LIN {X 0,Y 474.756,Z 198.653,A -85,B 0,C 180,E1 -7374.053,E2 -7374.053} C_VEL
LIN {X 0,Y 474.86,Z 198.632,A -85,B 0,C 180,E1 -7377.456,E2 -7377.456} C_VEL
LIN {X 0,Y 474.875,Z 198.64,A -85,B 0,C 180,E1 -7380,E2 -7380} C_VEL
LIN {X 0,Y 474.861,Z 198.647,A -85,B 0,C 180,E1 -7382.545,E2 -7382.545} C_VEL
LIN {X 0,Y 474.75,Z 198.651,A -85,B 0,C 180,E1 -7385.948,E2 -7385.948} C_VEL
LIN {X 0,Y 474.696,Z 198.67,A -85,B 0,C 180,E1 -7388.515,E2 -7388.515} C_VEL
LIN {X 0,Y 474.673,Z 198.655,A -85,B 0,C 180,E1 -7391.964,E2 -7391.964} C_VEL
LIN {X 0,Y 474.669,Z 198.666,A -85,B 0,C 180,E1 -7395.457,E2 -7395.457} C_VEL
LIN {X 0,Y 474.635,Z 198.663,A -85,B 0,C 180,E1 -7399.012,E2 -7399.012} C_VEL
LIN {X 0,Y 474.568,Z 198.678,A -85,B 0,C 180,E1 -7401.73,E2 -7401.73} C_VEL
LIN {X 0,Y 474.634,Z 198.67,A -85,B 0,C 180,E1 -7404.495,E2 -7404.495} C_VEL
LIN {X 0,Y 474.654,Z 198.664,A -85,B 0,C 180,E1 -7407.337,E2 -7407.337} C_VEL
LIN {X 0,Y 474.579,Z 198.684,A -85,B 0,C 180,E1 -7410.233,E2 -7410.233} C_VEL
LIN {X 0,Y 474.618,Z 198.665,A -85,B 0,C 180,E1 -7413.223,E2 -7413.223} C_VEL
LIN {X 0,Y 474.568,Z 198.687,A -85,B 0,C 180,E1 -7416.326,E2 -7416.326} C_VEL
LIN {X 0,Y 474.595,Z 198.667,A -85,B 0,C 180,E1 -7419.649,E2 -7419.649} C_VEL
LIN {X 0,Y 474.604,Z 198.682,A -85,B 0,C 180,E1 -7422.24,E2 -7422.24} C_VEL
LIN {X 0,Y 474.598,Z 198.667,A -85,B 0,C 180,E1 -7425.301,E2 -7425.301} C_VEL
LIN {X 0,Y 474.598,Z 198.682,A -85,B 0,C 180,E1 -7428.217,E2 -7428.217} C_VEL
LIN {X 0,Y 474.597,Z 198.672,A -85,B 0,C 180,E1 -7431.546,E2 -7431.546} C_VEL
LIN {X 0,Y 474.615,Z 198.669,A -85,B 0,C 180,E1 -7434.729,E2 -7434.729} C_VEL
LIN {X 0,Y 474.625,Z 198.676,A -85,B 0,C 180,E1 -7437.791,E2 -7437.791} C_VEL
LIN {X 0,Y 474.598,Z 198.675,A -85,B 0,C 180,E1 -7440.892,E2 -7440.892} C_VEL
LIN {X 0,Y 474.595,Z 198.679,A -85,B 0,C 180,E1 -7443.628,E2 -7443.628} C_VEL
LIN {X 0,Y 474.629,Z 198.672,A -85,B 0,C 180,E1 -7446.645,E2 -7446.645} C_VEL
LIN {X 0,Y 474.644,Z 198.673,A -85,B 0,C 180,E1 -7450.092,E2 -7450.092} C_VEL
LIN {X 0,Y 474.635,Z 198.675,A -85,B 0,C 180,E1 -7451.709,E2 -7451.709} C_VEL
LIN {X 0,Y 473.961,Z 198.765,A -85,B 0,C 180,E1 -7452.418,E2 -7452.418} C_VEL
LIN {X 0,Y 471.109,Z 199.122,A -85,B 0,C 180,E1 -7453.569,E2 -7453.569} C_VEL
LIN {X 0,Y 468.702,Z 199.417,A -85,B 0,C 180,E1 -7454.497,E2 -7454.497} C_VEL
LIN {X 0,Y 467.668,Z 199.542,A -85,B 0,C 180,E1 -7455.214,E2 -7455.214} C_VEL
LIN {X 0,Y 467.584,Z 199.551,A -85,B 0,C 180,E1 -7455.457,E2 -7455.457} C_VEL
LIN {X 0,Y 467.65,Z 199.543,A -85,B 0,C 180,E1 -7458.736,E2 -7458.736} C_VEL
LIN {X 0,Y 467.658,Z 199.545,A -85,B 0,C 180,E1 -7461.359,E2 -7461.359} C_VEL
LIN {X 0,Y 467.705,Z 199.531,A -85,B 0,C 180,E1 -7463.964,E2 -7463.964} C_VEL
LIN {X 0,Y 467.597,Z 199.662,A -85,B 0,C 180,E1 -7466.367,E2 -7466.367} C_VEL
LIN {X 0,Y 470.549,Z 209.002,A -85,B 0,C 180,E1 -7467.722,E2 -7467.722} C_VEL
LIN {X 0,Y 480.125,Z 229.823,A -85,B 0,C 180,E1 -7468.71,E2 -7468.71} C_VEL
LIN {X 0,Y 478.57,Z 337.497,A -85,B 0,C 180,E1 -7470.42,E2 -7470.42} C_VEL
LIN {X 0,Y 477.488,Z 414.636,A -85,B 0,C 180,E1 -7471.66,E2 -7471.66} C_VEL
LIN {X 0,Y 476.912,Z 431.039,A -85,B 0,C 180,E1 -7472.087,E2 -7472.087} C_VEL
LIN {X 0,Y 476.258,Z 446.341,A -85,B 0,C 180,E1 -7472.645,E2 -7472.645} C_VEL
LIN {X 0,Y 475.341,Z 462.22,A -85,B 0,C 180,E1 -7473.392,E2 -7473.392} C_VEL
LIN {X 0,Y 474.435,Z 476.76,A -85,B 0,C 180,E1 -7474.249,E2 -7474.249} C_VEL
LIN {X 0,Y 473.289,Z 491.411,A -85,B 0,C 180,E1 -7475.302,E2 -7475.302} C_VEL
LIN {X 0,Y 472.273,Z 504.308,A -85,B 0,C 180,E1 -7476.41,E2 -7476.41} C_VEL
LIN {X 0,Y 471.217,Z 517.245,A -85,B 0,C 180,E1 -7477.716,E2 -7477.716} C_VEL
LIN {X 0,Y 470.216,Z 529.305,A -85,B 0,C 180,E1 -7479.147,E2 -7479.147} C_VEL
LIN {X 0,Y 469.224,Z 540.984,A -85,B 0,C 180,E1 -7480.792,E2 -7480.792} C_VEL
LIN {X 0,Y 468.482,Z 550.373,A -85,B 0,C 180,E1 -7482.355,E2 -7482.355} C_VEL
LIN {X 0,Y 467.914,Z 559.42,A -85,B 0,C 180,E1 -7484.129,E2 -7484.129} C_VEL
LIN {X 0,Y 467.444,Z 566.588,A -85,B 0,C 180,E1 -7485.794,E2 -7485.794} C_VEL
LIN {X 0,Y 467.03,Z 574.14,A -85,B 0,C 180,E1 -7487.97,E2 -7487.97} C_VEL
LIN {X 0,Y 466.828,Z 579.053,A -85,B 0,C 180,E1 -7489.801,E2 -7489.801} C_VEL
LIN {X 0,Y 466.675,Z 582.05,A -85,B 0,C 180,E1 -7491.19,E2 -7491.19} C_VEL
LIN {X 0,Y 466.513,Z 585.196,A -85,B 0,C 180,E1 -7493.224,E2 -7493.224} C_VEL
LIN {X 0,Y 466.473,Z 587.043,A -85,B 0,C 180,E1 -7495.313,E2 -7495.313} C_VEL
LIN {X 0,Y 466.497,Z 587.539,A -85,B 0,C 180,E1 -7497.268,E2 -7497.268} C_VEL
LIN {X 0,Y 466.524,Z 586.882,A -85,B 0,C 180,E1 -7499.102,E2 -7499.102} C_VEL
LIN {X 0,Y 466.589,Z 585.259,A -85,B 0,C 180,E1 -7500.843,E2 -7500.843} C_VEL
LIN {X 0,Y 466.678,Z 582.245,A -85,B 0,C 180,E1 -7502.831,E2 -7502.831} C_VEL
LIN {X 0,Y 466.811,Z 579.574,A -85,B 0,C 180,E1 -7504.101,E2 -7504.101} C_VEL
LIN {X 0,Y 467.041,Z 574.75,A -85,B 0,C 180,E1 -7505.936,E2 -7505.936} C_VEL
LIN {X 0,Y 467.282,Z 569.408,A -85,B 0,C 180,E1 -7507.562,E2 -7507.562} C_VEL
LIN {X 0,Y 467.669,Z 563.253,A -85,B 0,C 180,E1 -7509.137,E2 -7509.137} C_VEL
LIN {X 0,Y 468.147,Z 555.633,A -85,B 0,C 180,E1 -7510.772,E2 -7510.772} C_VEL
LIN {X 0,Y 468.822,Z 546.607,A -85,B 0,C 180,E1 -7512.423,E2 -7512.423} C_VEL
LIN {X 0,Y 469.752,Z 535.757,A -85,B 0,C 180,E1 -7514.099,E2 -7514.099} C_VEL
LIN {X 0,Y 470.651,Z 524.675,A -85,B 0,C 180,E1 -7515.547,E2 -7515.547} C_VEL
LIN {X 0,Y 471.687,Z 512.615,A -85,B 0,C 180,E1 -7516.894,E2 -7516.894} C_VEL
LIN {X 0,Y 472.776,Z 499.201,A -85,B 0,C 180,E1 -7518.171,E2 -7518.171} C_VEL
LIN {X 0,Y 473.863,Z 485.577,A -85,B 0,C 180,E1 -7519.263,E2 -7519.263} C_VEL
LIN {X 0,Y 474.967,Z 469.802,A -85,B 0,C 180,E1 -7520.304,E2 -7520.304} C_VEL
LIN {X 0,Y 475.881,Z 455.142,A -85,B 0,C 180,E1 -7521.081,E2 -7521.081} C_VEL
LIN {X 0,Y 476.692,Z 438.798,A -85,B 0,C 180,E1 -7521.767,E2 -7521.767} C_VEL
LIN {X 0,Y 477.372,Z 422.454,A -85,B 0,C 180,E1 -7522.269,E2 -7522.269} C_VEL
LIN {X 0,Y 477.774,Z 405.589,A -85,B 0,C 180,E1 -7522.617,E2 -7522.617} C_VEL
LIN {X 0,Y 480.45,Z 230.253,A -85,B 0,C 180,E1 -7525.405,E2 -7525.405} C_VEL
LIN {X 0,Y 471.765,Z 211.838,A -85,B 0,C 180,E1 -7526.32,E2 -7526.32} C_VEL
LIN {X 0,Y 470.58,Z 209.292,A -85,B 0,C 180,E1 -7526.455,E2 -7526.455} C_VEL
LIN {X 0,Y 467.6,Z 199.551,A -85,B 0,C 180,E1 -7527.944,E2 -7527.944} C_VEL
LIN {X 0,Y 467.579,Z 199.553,A -85,B 0,C 180,E1 -7531.25,E2 -7531.25} C_VEL
LIN {X 0,Y 467.599,Z 199.551,A -85,B 0,C 180,E1 -7534.159,E2 -7534.159} C_VEL
LIN {X 0,Y 467.577,Z 199.554,A -85,B 0,C 180,E1 -7536.995,E2 -7536.995} C_VEL
LIN {X 0,Y 467.624,Z 199.545,A -85,B 0,C 180,E1 -7539.777,E2 -7539.777} C_VEL
LIN {X 0,Y 467.609,Z 199.543,A -85,B 0,C 180,E1 -7542.506,E2 -7542.506} C_VEL
LIN {X 0,Y 467.606,Z 199.548,A -85,B 0,C 180,E1 -7545.196,E2 -7545.196} C_VEL
LIN {X 0,Y 467.656,Z 199.546,A -85,B 0,C 180,E1 -7547.854,E2 -7547.854} C_VEL
LIN {X 0,Y 467.679,Z 199.541,A -85,B 0,C 180,E1 -7551.357,E2 -7551.357} C_VEL
LIN {X 0,Y 467.741,Z 199.534,A -85,B 0,C 180,E1 -7553.962,E2 -7553.962} C_VEL
LIN {X 0,Y 467.856,Z 199.518,A -85,B 0,C 180,E1 -7557.417,E2 -7557.417} C_VEL
LIN {X 0,Y 467.879,Z 199.518,A -85,B 0,C 180,E1 -7560,E2 -7560} C_VEL
LIN {X 0,Y 467.855,Z 199.516,A -85,B 0,C 180,E1 -7562.582,E2 -7562.582} C_VEL
LIN {X 0,Y 467.731,Z 199.534,A -85,B 0,C 180,E1 -7566.037,E2 -7566.037} C_VEL
LIN {X 0,Y 467.668,Z 199.54,A -85,B 0,C 180,E1 -7568.643,E2 -7568.643} C_VEL
LIN {X 0,Y 467.654,Z 199.542,A -85,B 0,C 180,E1 -7572.145,E2 -7572.145} C_VEL
LIN {X 0,Y 467.637,Z 199.545,A -85,B 0,C 180,E1 -7575.695,E2 -7575.695} C_VEL
LIN {X 0,Y 467.62,Z 199.548,A -85,B 0,C 180,E1 -7579.307,E2 -7579.307} C_VEL
LIN {X 0,Y 467.532,Z 199.556,A -85,B 0,C 180,E1 -7582.074,E2 -7582.074} C_VEL
LIN {X 0,Y 467.583,Z 199.55,A -85,B 0,C 180,E1 -7584.888,E2 -7584.888} C_VEL
LIN {X 0,Y 467.618,Z 199.548,A -85,B 0,C 180,E1 -7587.769,E2 -7587.769} C_VEL
LIN {X 0,Y 467.566,Z 199.558,A -85,B 0,C 180,E1 -7591.044,E2 -7591.044} C_VEL
LIN {X 0,Y 467.576,Z 199.55,A -85,B 0,C 180,E1 -7594.239,E2 -7594.239} C_VEL
LIN {X 0,Y 467.547,Z 199.561,A -85,B 0,C 180,E1 -7597.186,E2 -7597.186} C_VEL
LIN {X 0,Y 467.57,Z 199.552,A -85,B 0,C 180,E1 -7600.265,E2 -7600.265} C_VEL
LIN {X 0,Y 467.548,Z 199.555,A -85,B 0,C 180,E1 -7603.745,E2 -7603.745} C_VEL
LIN {X 0,Y 467.547,Z 199.56,A -85,B 0,C 180,E1 -7606.254,E2 -7606.254} C_VEL
LIN {X 0,Y 467.56,Z 199.555,A -85,B 0,C 180,E1 -7609.733,E2 -7609.733} C_VEL
LIN {X 0,Y 467.543,Z 199.557,A -85,B 0,C 180,E1 -7612.814,E2 -7612.814} C_VEL
LIN {X 0,Y 467.585,Z 199.552,A -85,B 0,C 180,E1 -7616.211,E2 -7616.211} C_VEL
LIN {X 0,Y 467.622,Z 199.679,A -85,B 0,C 180,E1 -7616.715,E2 -7616.715} C_VEL
LIN {X 0,Y 473.66,Z 219.016,A -85,B 0,C 180,E1 -7619.381,E2 -7619.381} C_VEL
LIN {X 0,Y 475.873,Z 227.663,A -85,B 0,C 180,E1 -7620.491,E2 -7620.491} C_VEL
LIN {X 0,Y 475.592,Z 231.809,A -85,B 0,C 180,E1 -7620.928,E2 -7620.928} C_VEL
LIN {X 0,Y 480.062,Z 257.211,A -85,B 0,C 180,E1 -7621.668,E2 -7621.668} C_VEL
LIN {X 0,Y 478.274,Z 376.342,A -85,B 0,C 180,E1 -7623.564,E2 -7623.564} C_VEL
LIN {X 0,Y 477.338,Z 440.054,A -85,B 0,C 180,E1 -7624.595,E2 -7624.595} C_VEL
LIN {X 0,Y 476.616,Z 457.299,A -85,B 0,C 180,E1 -7625.047,E2 -7625.047} C_VEL
LIN {X 0,Y 475.877,Z 472.946,A -85,B 0,C 180,E1 -7625.631,E2 -7625.631} C_VEL
LIN {X 0,Y 474.949,Z 487.77,A -85,B 0,C 180,E1 -7626.334,E2 -7626.334} C_VEL
LIN {X 0,Y 473.975,Z 502.298,A -85,B 0,C 180,E1 -7627.187,E2 -7627.187} C_VEL
LIN {X 0,Y 472.892,Z 516.304,A -85,B 0,C 180,E1 -7628.188,E2 -7628.188} C_VEL
LIN {X 0,Y 471.72,Z 530.44,A -85,B 0,C 180,E1 -7629.39,E2 -7629.39} C_VEL
LIN {X 0,Y 470.682,Z 542.772,A -85,B 0,C 180,E1 -7630.625,E2 -7630.625} C_VEL
LIN {X 0,Y 469.688,Z 555.582,A -85,B 0,C 180,E1 -7632.135,E2 -7632.135} C_VEL
LIN {X 0,Y 468.773,Z 567.224,A -85,B 0,C 180,E1 -7633.762,E2 -7633.762} C_VEL
LIN {X 0,Y 468.157,Z 576.066,A -85,B 0,C 180,E1 -7635.213,E2 -7635.213} C_VEL
LIN {X 0,Y 467.611,Z 585.271,A -85,B 0,C 180,E1 -7636.969,E2 -7636.969} C_VEL
LIN {X 0,Y 467.2,Z 592.974,A -85,B 0,C 180,E1 -7638.721,E2 -7638.721} C_VEL
LIN {X 0,Y 466.853,Z 600.714,A -85,B 0,C 180,E1 -7640.904,E2 -7640.904} C_VEL
LIN {X 0,Y 466.772,Z 605.522,A -85,B 0,C 180,E1 -7642.645,E2 -7642.645} C_VEL
LIN {X 0,Y 466.697,Z 608.448,A -85,B 0,C 180,E1 -7643.947,E2 -7643.947} C_VEL
LIN {X 0,Y 466.599,Z 611.421,A -85,B 0,C 180,E1 -7645.679,E2 -7645.679} C_VEL
LIN {X 0,Y 466.651,Z 613.381,A -85,B 0,C 180,E1 -7647.408,E2 -7647.408} C_VEL
LIN {X 0,Y 466.615,Z 614.357,A -85,B 0,C 180,E1 -7649.135,E2 -7649.135} C_VEL
LIN {X 0,Y 466.615,Z 614.365,A -85,B 0,C 180,E1 -7650.861,E2 -7650.861} C_VEL
LIN {X 0,Y 466.65,Z 613.404,A -85,B 0,C 180,E1 -7652.587,E2 -7652.587} C_VEL
LIN {X 0,Y 466.598,Z 611.461,A -85,B 0,C 180,E1 -7654.317,E2 -7654.317} C_VEL
LIN {X 0,Y 466.746,Z 607.794,A -85,B 0,C 180,E1 -7656.391,E2 -7656.391} C_VEL
LIN {X 0,Y 466.79,Z 603.336,A -85,B 0,C 180,E1 -7658.221,E2 -7658.221} C_VEL
LIN {X 0,Y 466.969,Z 597.932,A -85,B 0,C 180,E1 -7659.964,E2 -7659.964} C_VEL
LIN {X 0,Y 467.336,Z 591.264,A -85,B 0,C 180,E1 -7661.711,E2 -7661.711} C_VEL
LIN {X 0,Y 467.733,Z 583.271,A -85,B 0,C 180,E1 -7663.465,E2 -7663.465} C_VEL
LIN {X 0,Y 468.419,Z 573.731,A -85,B 0,C 180,E1 -7665.22,E2 -7665.22} C_VEL
LIN {X 0,Y 469.184,Z 562.298,A -85,B 0,C 180,E1 -7666.981,E2 -7666.981} C_VEL
LIN {X 0,Y 470.161,Z 550.414,A -85,B 0,C 180,E1 -7668.518,E2 -7668.518} C_VEL
LIN {X 0,Y 471.123,Z 538.265,A -85,B 0,C 180,E1 -7669.861,E2 -7669.861} C_VEL
LIN {X 0,Y 472.265,Z 524.529,A -85,B 0,C 180,E1 -7671.151,E2 -7671.151} C_VEL
LIN {X 0,Y 473.318,Z 510.73,A -85,B 0,C 180,E1 -7672.246,E2 -7672.246} C_VEL
LIN {X 0,Y 474.473,Z 494.982,A -85,B 0,C 180,E1 -7673.27,E2 -7673.27} C_VEL
LIN {X 0,Y 475.417,Z 480.293,A -85,B 0,C 180,E1 -7674.042,E2 -7674.042} C_VEL
LIN {X 0,Y 476.317,Z 463.971,A -85,B 0,C 180,E1 -7674.718,E2 -7674.718} C_VEL
LIN {X 0,Y 476.985,Z 448.256,A -85,B 0,C 180,E1 -7675.205,E2 -7675.205} C_VEL
LIN {X 0,Y 477.512,Z 431.69,A -85,B 0,C 180,E1 -7675.546,E2 -7675.546} C_VEL
LIN {X 0,Y 479.984,Z 258.583,A -85,B 0,C 180,E1 -7678.281,E2 -7678.281} C_VEL
LIN {X 0,Y 478.559,Z 248.971,A -85,B 0,C 180,E1 -7678.534,E2 -7678.534} C_VEL
LIN {X 0,Y 475.596,Z 232.132,A -85,B 0,C 180,E1 -7679.039,E2 -7679.039} C_VEL
LIN {X 0,Y 475.884,Z 227.612,A -85,B 0,C 180,E1 -7679.514,E2 -7679.514} C_VEL
LIN {X 0,Y 472.324,Z 214.704,A -85,B 0,C 180,E1 -7681.178,E2 -7681.178} C_VEL
LIN {X 0,Y 467.604,Z 199.536,A -85,B 0,C 180,E1 -7683.266,E2 -7683.266} C_VEL
LIN {X 0,Y 467.536,Z 199.56,A -85,B 0,C 180,E1 -7685.887,E2 -7685.887} C_VEL
LIN {X 0,Y 467.556,Z 199.559,A -85,B 0,C 180,E1 -7689.143,E2 -7689.143} C_VEL
LIN {X 0,Y 467.565,Z 199.552,A -85,B 0,C 180,E1 -7692.565,E2 -7692.565} C_VEL
LIN {X 0,Y 467.547,Z 199.556,A -85,B 0,C 180,E1 -7695.051,E2 -7695.051} C_VEL
LIN {X 0,Y 467.565,Z 199.557,A -85,B 0,C 180,E1 -7697.438,E2 -7697.438} C_VEL
LIN {X 0,Y 467.587,Z 199.553,A -85,B 0,C 180,E1 -7700.856,E2 -7700.856} C_VEL
LIN {X 0,Y 467.535,Z 199.552,A -85,B 0,C 180,E1 -7704.258,E2 -7704.258} C_VEL
LIN {X 0,Y 467.554,Z 199.548,A -85,B 0,C 180,E1 -7707.319,E2 -7707.319} C_VEL
LIN {X 0,Y 467.54,Z 199.559,A -85,B 0,C 180,E1 -7710.666,E2 -7710.666} C_VEL
LIN {X 0,Y 467.585,Z 199.542,A -85,B 0,C 180,E1 -7713.198,E2 -7713.198} C_VEL
LIN {X 0,Y 467.566,Z 199.554,A -85,B 0,C 180,E1 -7716.466,E2 -7716.466} C_VEL
LIN {X 0,Y 467.594,Z 199.536,A -85,B 0,C 180,E1 -7719.776,E2 -7719.776} C_VEL
LIN {X 0,Y 467.576,Z 199.549,A -85,B 0,C 180,E1 -7722.506,E2 -7722.506} C_VEL
LIN {X 0,Y 467.573,Z 199.549,A -85,B 0,C 180,E1 -7725.196,E2 -7725.196} C_VEL
LIN {X 0,Y 467.65,Z 199.521,A -85,B 0,C 180,E1 -7727.855,E2 -7727.855} C_VEL
LIN {X 0,Y 467.65,Z 199.543,A -85,B 0,C 180,E1 -7731.357,E2 -7731.357} C_VEL
LIN {X 0,Y 467.718,Z 199.529,A -85,B 0,C 180,E1 -7733.963,E2 -7733.963} C_VEL
LIN {X 0,Y 467.826,Z 199.508,A -85,B 0,C 180,E1 -7737.417,E2 -7737.417} C_VEL
LIN {X 0,Y 467.846,Z 199.516,A -85,B 0,C 180,E1 -7740,E2 -7740} C_VEL
LIN {X 0,Y 467.826,Z 199.522,A -85,B 0,C 180,E1 -7742.584,E2 -7742.584} C_VEL
LIN {X 0,Y 467.714,Z 199.528,A -85,B 0,C 180,E1 -7746.038,E2 -7746.038} C_VEL
LIN {X 0,Y 467.65,Z 199.546,A -85,B 0,C 180,E1 -7748.644,E2 -7748.644} C_VEL
LIN {X 0,Y 467.624,Z 199.534,A -85,B 0,C 180,E1 -7752.147,E2 -7752.147} C_VEL
LIN {X 0,Y 467.624,Z 199.544,A -85,B 0,C 180,E1 -7755.696,E2 -7755.696} C_VEL
LIN {X 0,Y 467.587,Z 199.541,A -85,B 0,C 180,E1 -7758.766,E2 -7758.766} C_VEL
LIN {X 0,Y 467.554,Z 199.552,A -85,B 0,C 180,E1 -7761.271,E2 -7761.271} C_VEL
LIN {X 0,Y 467.547,Z 199.555,A -85,B 0,C 180,E1 -7763.945,E2 -7763.945} C_VEL
LIN {X 0,Y 467.589,Z 199.547,A -85,B 0,C 180,E1 -7766.803,E2 -7766.803} C_VEL
LIN {X 0,Y 467.527,Z 199.558,A -85,B 0,C 180,E1 -7769.741,E2 -7769.741} C_VEL
LIN {X 0,Y 467.558,Z 199.546,A -85,B 0,C 180,E1 -7772.761,E2 -7772.761} C_VEL
LIN {X 0,Y 467.532,Z 199.558,A -85,B 0,C 180,E1 -7775.892,E2 -7775.892} C_VEL
LIN {X 0,Y 467.537,Z 199.544,A -85,B 0,C 180,E1 -7779.15,E2 -7779.15} C_VEL
LIN {X 0,Y 467.567,Z 199.555,A -85,B 0,C 180,E1 -7782.57,E2 -7782.57} C_VEL
LIN {X 0,Y 467.547,Z 199.545,A -85,B 0,C 180,E1 -7785.055,E2 -7785.055} C_VEL
LIN {X 0,Y 467.557,Z 199.554,A -85,B 0,C 180,E1 -7788.6,E2 -7788.6} C_VEL
LIN {X 0,Y 467.551,Z 199.554,A -85,B 0,C 180,E1 -7791.959,E2 -7791.959} C_VEL
LIN {X 0,Y 467.554,Z 199.547,A -85,B 0,C 180,E1 -7795.171,E2 -7795.171} C_VEL
LIN {X 0,Y 467.572,Z 199.556,A -85,B 0,C 180,E1 -7798.263,E2 -7798.263} C_VEL
LIN {X 0,Y 467.546,Z 199.553,A -85,B 0,C 180,E1 -7801.252,E2 -7801.252} C_VEL
LIN {X 0,Y 467.572,Z 199.552,A -85,B 0,C 180,E1 -7804.161,E2 -7804.161} C_VEL
LIN {X 0,Y 467.57,Z 199.55,A -85,B 0,C 180,E1 -7806.999,E2 -7806.999} C_VEL
LIN {X 0,Y 467.615,Z 199.553,A -85,B 0,C 180,E1 -7809.78,E2 -7809.78} C_VEL
LIN {X 0,Y 467.565,Z 199.555,A -85,B 0,C 180,E1 -7812.508,E2 -7812.508} C_VEL
LIN {X 0,Y 467.584,Z 199.551,A -85,B 0,C 180,E1 -7815.457,E2 -7815.457} C_VEL
LIN {X 0,Y 466.918,Z 199.636,A -85,B 0,C 180,E1 -7816.176,E2 -7816.176} C_VEL
LIN {X 0,Y 464.078,Z 199.99,A -85,B 0,C 180,E1 -7817.345,E2 -7817.345} C_VEL
LIN {X 0,Y 461.68,Z 200.288,A -85,B 0,C 180,E1 -7818.287,E2 -7818.287} C_VEL
LIN {X 0,Y 460.653,Z 200.415,A -85,B 0,C 180,E1 -7819.015,E2 -7819.015} C_VEL
LIN {X 0,Y 460.571,Z 200.426,A -85,B 0,C 180,E1 -7819.261,E2 -7819.261} C_VEL
LIN {X 0,Y 460.666,Z 200.416,A -85,B 0,C 180,E1 -7822.596,E2 -7822.596} C_VEL
LIN {X 0,Y 460.677,Z 200.403,A -85,B 0,C 180,E1 -7824.75,E2 -7824.75} C_VEL
LIN {X 0,Y 460.553,Z 200.62,A -85,B 0,C 180,E1 -7825.955,E2 -7825.955} C_VEL
LIN {X 0,Y 463.312,Z 209.012,A -85,B 0,C 180,E1 -7827.225,E2 -7827.225} C_VEL
LIN {X 0,Y 473.85,Z 231.782,A -85,B 0,C 180,E1 -7828.337,E2 -7828.337} C_VEL
LIN {X 0,Y 472.34,Z 332.526,A -85,B 0,C 180,E1 -7829.962,E2 -7829.962} C_VEL
LIN {X 0,Y 471.041,Z 415.463,A -85,B 0,C 180,E1 -7831.311,E2 -7831.311} C_VEL
LIN {X 0,Y 470.43,Z 432.452,A -85,B 0,C 180,E1 -7831.768,E2 -7831.768} C_VEL
LIN {X 0,Y 469.701,Z 448.061,A -85,B 0,C 180,E1 -7832.36,E2 -7832.36} C_VEL
LIN {X 0,Y 468.723,Z 463.616,A -85,B 0,C 180,E1 -7833.118,E2 -7833.118} C_VEL
LIN {X 0,Y 467.764,Z 477.967,A -85,B 0,C 180,E1 -7833.987,E2 -7833.987} C_VEL
LIN {X 0,Y 466.566,Z 492.8,A -85,B 0,C 180,E1 -7835.079,E2 -7835.079} C_VEL
LIN {X 0,Y 465.442,Z 506.377,A -85,B 0,C 180,E1 -7836.287,E2 -7836.287} C_VEL
LIN {X 0,Y 464.298,Z 519.039,A -85,B 0,C 180,E1 -7837.613,E2 -7837.613} C_VEL
LIN {X 0,Y 463.321,Z 530.181,A -85,B 0,C 180,E1 -7838.973,E2 -7838.973} C_VEL
LIN {X 0,Y 462.372,Z 540.923,A -85,B 0,C 180,E1 -7840.511,E2 -7840.511} C_VEL
LIN {X 0,Y 461.575,Z 550.304,A -85,B 0,C 180,E1 -7842.086,E2 -7842.086} C_VEL
LIN {X 0,Y 460.928,Z 559.45,A -85,B 0,C 180,E1 -7843.897,E2 -7843.897} C_VEL
LIN {X 0,Y 460.452,Z 566.134,A -85,B 0,C 180,E1 -7845.463,E2 -7845.463} C_VEL
LIN {X 0,Y 460.041,Z 572.746,A -85,B 0,C 180,E1 -7847.333,E2 -7847.333} C_VEL
LIN {X 0,Y 459.826,Z 578.038,A -85,B 0,C 180,E1 -7849.186,E2 -7849.186} C_VEL
LIN {X 0,Y 459.592,Z 582.296,A -85,B 0,C 180,E1 -7851.123,E2 -7851.123} C_VEL
LIN {X 0,Y 459.435,Z 584.534,A -85,B 0,C 180,E1 -7852.485,E2 -7852.485} C_VEL
LIN {X 0,Y 459.375,Z 586.654,A -85,B 0,C 180,E1 -7854.399,E2 -7854.399} C_VEL
LIN {X 0,Y 459.372,Z 587.654,A -85,B 0,C 180,E1 -7856.34,E2 -7856.34} C_VEL
LIN {X 0,Y 459.413,Z 587.529,A -85,B 0,C 180,E1 -7858.31,E2 -7858.31} C_VEL
LIN {X 0,Y 459.456,Z 586.119,A -85,B 0,C 180,E1 -7860.318,E2 -7860.318} C_VEL
LIN {X 0,Y 459.542,Z 583.383,A -85,B 0,C 180,E1 -7862.363,E2 -7862.363} C_VEL
LIN {X 0,Y 459.748,Z 579.221,A -85,B 0,C 180,E1 -7864.445,E2 -7864.445} C_VEL
LIN {X 0,Y 460.052,Z 573.451,A -85,B 0,C 180,E1 -7866.57,E2 -7866.57} C_VEL
LIN {X 0,Y 460.422,Z 566.932,A -85,B 0,C 180,E1 -7868.465,E2 -7868.465} C_VEL
LIN {X 0,Y 460.963,Z 559.007,A -85,B 0,C 180,E1 -7870.33,E2 -7870.33} C_VEL
LIN {X 0,Y 461.624,Z 550.21,A -85,B 0,C 180,E1 -7872.058,E2 -7872.058} C_VEL
LIN {X 0,Y 462.534,Z 540.105,A -85,B 0,C 180,E1 -7873.738,E2 -7873.738} C_VEL
LIN {X 0,Y 463.467,Z 528.983,A -85,B 0,C 180,E1 -7875.314,E2 -7875.314} C_VEL
LIN {X 0,Y 464.666,Z 516.026,A -85,B 0,C 180,E1 -7876.86,E2 -7876.86} C_VEL
LIN {X 0,Y 465.903,Z 502.305,A -85,B 0,C 180,E1 -7878.23,E2 -7878.23} C_VEL
LIN {X 0,Y 467.106,Z 487.756,A -85,B 0,C 180,E1 -7879.443,E2 -7879.443} C_VEL
LIN {X 0,Y 468.235,Z 473.076,A -85,B 0,C 180,E1 -7880.455,E2 -7880.455} C_VEL
LIN {X 0,Y 469.238,Z 457.631,A -85,B 0,C 180,E1 -7881.325,E2 -7881.325} C_VEL
LIN {X 0,Y 470.082,Z 443.266,A -85,B 0,C 180,E1 -7881.972,E2 -7881.972} C_VEL
LIN {X 0,Y 470.812,Z 426.598,A -85,B 0,C 180,E1 -7882.535,E2 -7882.535} C_VEL
LIN {X 0,Y 471.289,Z 410.62,A -85,B 0,C 180,E1 -7882.905,E2 -7882.905} C_VEL
LIN {X 0,Y 474.22,Z 232.357,A -85,B 0,C 180,E1 -7885.789,E2 -7885.789} C_VEL
LIN {X 0,Y 465.202,Z 213.206,A -85,B 0,C 180,E1 -7886.767,E2 -7886.767} C_VEL
LIN {X 0,Y 463.377,Z 209.586,A -85,B 0,C 180,E1 -7886.971,E2 -7886.971} C_VEL
LIN {X 0,Y 460.549,Z 200.43,A -85,B 0,C 180,E1 -7888.409,E2 -7888.409} C_VEL
LIN {X 0,Y 460.555,Z 200.427,A -85,B 0,C 180,E1 -7891.767,E2 -7891.767} C_VEL
LIN {X 0,Y 460.541,Z 200.434,A -85,B 0,C 180,E1 -7894.704,E2 -7894.704} C_VEL
LIN {X 0,Y 460.512,Z 200.436,A -85,B 0,C 180,E1 -7897.571,E2 -7897.571} C_VEL
LIN {X 0,Y 460.57,Z 200.43,A -85,B 0,C 180,E1 -7900.384,E2 -7900.384} C_VEL
LIN {X 0,Y 460.566,Z 200.421,A -85,B 0,C 180,E1 -7903.146,E2 -7903.146} C_VEL
LIN {X 0,Y 460.554,Z 200.43,A -85,B 0,C 180,E1 -7905.867,E2 -7905.867} C_VEL
LIN {X 0,Y 460.609,Z 200.42,A -85,B 0,C 180,E1 -7908.559,E2 -7908.559} C_VEL
LIN {X 0,Y 460.695,Z 200.414,A -85,B 0,C 180,E1 -7912.108,E2 -7912.108} C_VEL
LIN {X 0,Y 460.694,Z 200.409,A -85,B 0,C 180,E1 -7914.748,E2 -7914.748} C_VEL
LIN {X 0,Y 460.797,Z 200.397,A -85,B 0,C 180,E1 -7917.377,E2 -7917.377} C_VEL
LIN {X 0,Y 460.85,Z 200.394,A -85,B 0,C 180,E1 -7920,E2 -7920} C_VEL
LIN {X 0,Y 460.797,Z 200.396,A -85,B 0,C 180,E1 -7922.622,E2 -7922.622} C_VEL
LIN {X 0,Y 460.696,Z 200.41,A -85,B 0,C 180,E1 -7926.13,E2 -7926.13} C_VEL
LIN {X 0,Y 460.618,Z 200.418,A -85,B 0,C 180,E1 -7928.776,E2 -7928.776} C_VEL
LIN {X 0,Y 460.607,Z 200.419,A -85,B 0,C 180,E1 -7932.334,E2 -7932.334} C_VEL
LIN {X 0,Y 460.6,Z 200.42,A -85,B 0,C 180,E1 -7935.997,E2 -7935.997} C_VEL
LIN {X 0,Y 460.566,Z 200.429,A -85,B 0,C 180,E1 -7939.615,E2 -7939.615} C_VEL
LIN {X 0,Y 460.508,Z 200.43,A -85,B 0,C 180,E1 -7942.428,E2 -7942.428} C_VEL
LIN {X 0,Y 460.551,Z 200.428,A -85,B 0,C 180,E1 -7945.797,E2 -7945.797} C_VEL
LIN {X 0,Y 460.55,Z 200.427,A -85,B 0,C 180,E1 -7948.233,E2 -7948.233} C_VEL
LIN {X 0,Y 460.519,Z 200.434,A -85,B 0,C 180,E1 -7951.282,E2 -7951.282} C_VEL
LIN {X 0,Y 460.522,Z 200.429,A -85,B 0,C 180,E1 -7954.503,E2 -7954.503} C_VEL
LIN {X 0,Y 460.5,Z 200.434,A -85,B 0,C 180,E1 -7957.623,E2 -7957.623} C_VEL
LIN {X 0,Y 460.534,Z 200.429,A -85,B 0,C 180,E1 -7960.268,E2 -7960.268} C_VEL
LIN {X 0,Y 460.508,Z 200.435,A -85,B 0,C 180,E1 -7963.374,E2 -7963.374} C_VEL
LIN {X 0,Y 460.503,Z 200.44,A -85,B 0,C 180,E1 -7966.624,E2 -7966.624} C_VEL
LIN {X 0,Y 460.526,Z 200.431,A -85,B 0,C 180,E1 -7969.732,E2 -7969.732} C_VEL
LIN {X 0,Y 460.497,Z 200.434,A -85,B 0,C 180,E1 -7972.524,E2 -7972.524} C_VEL
LIN {X 0,Y 460.547,Z 200.431,A -85,B 0,C 180,E1 -7975.623,E2 -7975.623} C_VEL
LIN {X 0,Y 460.578,Z 200.535,A -85,B 0,C 180,E1 -7976.246,E2 -7976.246} C_VEL
LIN {X 0,Y 466.068,Z 217.829,A -85,B 0,C 180,E1 -7978.705,E2 -7978.705} C_VEL
LIN {X 0,Y 469.121,Z 228.633,A -85,B 0,C 180,E1 -7980.148,E2 -7980.148} C_VEL
LIN {X 0,Y 469.178,Z 231.798,A -85,B 0,C 180,E1 -7980.49,E2 -7980.49} C_VEL
LIN {X 0,Y 473.834,Z 258.34,A -85,B 0,C 180,E1 -7981.276,E2 -7981.276} C_VEL
LIN {X 0,Y 472.131,Z 363.89,A -85,B 0,C 180,E1 -7982.979,E2 -7982.979} C_VEL
LIN {X 0,Y 470.97,Z 438.936,A -85,B 0,C 180,E1 -7984.206,E2 -7984.206} C_VEL
LIN {X 0,Y 470.23,Z 455.754,A -85,B 0,C 180,E1 -7984.64,E2 -7984.64} C_VEL
LIN {X 0,Y 469.455,Z 471.44,A -85,B 0,C 180,E1 -7985.216,E2 -7985.216} C_VEL
LIN {X 0,Y 468.387,Z 487.561,A -85,B 0,C 180,E1 -7985.982,E2 -7985.982} C_VEL
LIN {X 0,Y 467.385,Z 502.31,A -85,B 0,C 180,E1 -7986.862,E2 -7986.862} C_VEL
LIN {X 0,Y 466.191,Z 516.083,A -85,B 0,C 180,E1 -7987.858,E2 -7987.858} C_VEL
LIN {X 0,Y 464.965,Z 530.214,A -85,B 0,C 180,E1 -7989.077,E2 -7989.077} C_VEL
LIN {X 0,Y 463.889,Z 542.737,A -85,B 0,C 180,E1 -7990.351,E2 -7990.351} C_VEL
LIN {X 0,Y 462.821,Z 555.359,A -85,B 0,C 180,E1 -7991.861,E2 -7991.861} C_VEL
LIN {X 0,Y 461.878,Z 566.634,A -85,B 0,C 180,E1 -7993.458,E2 -7993.458} C_VEL
LIN {X 0,Y 461.19,Z 575.842,A -85,B 0,C 180,E1 -7994.984,E2 -7994.984} C_VEL
LIN {X 0,Y 460.577,Z 585.049,A -85,B 0,C 180,E1 -7996.767,E2 -7996.767} C_VEL
LIN {X 0,Y 460.165,Z 592.756,A -85,B 0,C 180,E1 -7998.546,E2 -7998.546} C_VEL
LIN {X 0,Y 459.777,Z 600.499,A -85,B 0,C 180,E1 -8000.762,E2 -8000.762} C_VEL
LIN {X 0,Y 459.648,Z 606.392,A -85,B 0,C 180,E1 -8002.972,E2 -8002.972} C_VEL
LIN {X 0,Y 459.578,Z 609.843,A -85,B 0,C 180,E1 -8004.734,E2 -8004.734} C_VEL
LIN {X 0,Y 459.531,Z 612.351,A -85,B 0,C 180,E1 -8006.491,E2 -8006.491} C_VEL
LIN {X 0,Y 459.537,Z 613.771,A -85,B 0,C 180,E1 -8008.245,E2 -8008.245} C_VEL
LIN {X 0,Y 459.525,Z 614.311,A -85,B 0,C 180,E1 -8009.998,E2 -8009.998} C_VEL
LIN {X 0,Y 459.536,Z 613.788,A -85,B 0,C 180,E1 -8011.751,E2 -8011.751} C_VEL
LIN {X 0,Y 459.529,Z 612.385,A -85,B 0,C 180,E1 -8013.505,E2 -8013.505} C_VEL
LIN {X 0,Y 459.576,Z 609.895,A -85,B 0,C 180,E1 -8015.262,E2 -8015.262} C_VEL
LIN {X 0,Y 459.644,Z 606.466,A -85,B 0,C 180,E1 -8017.024,E2 -8017.024} C_VEL
LIN {X 0,Y 459.782,Z 600.596,A -85,B 0,C 180,E1 -8019.233,E2 -8019.233} C_VEL
LIN {X 0,Y 460.168,Z 592.872,A -85,B 0,C 180,E1 -8021.449,E2 -8021.449} C_VEL
LIN {X 0,Y 460.644,Z 584.16,A -85,B 0,C 180,E1 -8023.451,E2 -8023.451} C_VEL
LIN {X 0,Y 461.343,Z 574.751,A -85,B 0,C 180,E1 -8025.232,E2 -8025.232} C_VEL
LIN {X 0,Y 462.059,Z 565.056,A -85,B 0,C 180,E1 -8026.795,E2 -8026.795} C_VEL
LIN {X 0,Y 462.972,Z 553.756,A -85,B 0,C 180,E1 -8028.357,E2 -8028.357} C_VEL
LIN {X 0,Y 464.058,Z 541.342,A -85,B 0,C 180,E1 -8029.817,E2 -8029.817} C_VEL
LIN {X 0,Y 465.179,Z 527.995,A -85,B 0,C 180,E1 -8031.141,E2 -8031.141} C_VEL
LIN {X 0,Y 466.292,Z 514.754,A -85,B 0,C 180,E1 -8032.249,E2 -8032.249} C_VEL
LIN {X 0,Y 467.503,Z 500.502,A -85,B 0,C 180,E1 -8033.251,E2 -8033.251} C_VEL
LIN {X 0,Y 468.556,Z 485.557,A -85,B 0,C 180,E1 -8034.122,E2 -8034.122} C_VEL
LIN {X 0,Y 469.486,Z 470.014,A -85,B 0,C 180,E1 -8034.837,E2 -8034.837} C_VEL
LIN {X 0,Y 470.286,Z 453.552,A -85,B 0,C 180,E1 -8035.412,E2 -8035.412} C_VEL
LIN {X 0,Y 470.974,Z 436.801,A -85,B 0,C 180,E1 -8035.813,E2 -8035.813} C_VEL
LIN {X 0,Y 473.707,Z 259.506,A -85,B 0,C 180,E1 -8038.666,E2 -8038.666} C_VEL
LIN {X 0,Y 471.514,Z 245.825,A -85,B 0,C 180,E1 -8039.044,E2 -8039.044} C_VEL
LIN {X 0,Y 469.11,Z 232.22,A -85,B 0,C 180,E1 -8039.442,E2 -8039.442} C_VEL
LIN {X 0,Y 469.257,Z 229.83,A -85,B 0,C 180,E1 -8039.698,E2 -8039.698} C_VEL
LIN {X 0,Y 466.371,Z 219.094,A -85,B 0,C 180,E1 -8041.094,E2 -8041.094} C_VEL
LIN {X 0,Y 460.528,Z 200.422,A -85,B 0,C 180,E1 -8043.681,E2 -8043.681} C_VEL
LIN {X 0,Y 460.458,Z 200.443,A -85,B 0,C 180,E1 -8046.527,E2 -8046.527} C_VEL
LIN {X 0,Y 460.507,Z 200.43,A -85,B 0,C 180,E1 -8049.86,E2 -8049.86} C_VEL
LIN {X 0,Y 460.491,Z 200.433,A -85,B 0,C 180,E1 -8052.898,E2 -8052.898} C_VEL
LIN {X 0,Y 460.497,Z 200.431,A -85,B 0,C 180,E1 -8055.827,E2 -8055.827} C_VEL
LIN {X 0,Y 460.517,Z 200.43,A -85,B 0,C 180,E1 -8058.988,E2 -8058.988} C_VEL
LIN {X 0,Y 460.516,Z 200.436,A -85,B 0,C 180,E1 -8061.266,E2 -8061.266} C_VEL
LIN {X 0,Y 460.486,Z 200.432,A -85,B 0,C 180,E1 -8064.553,E2 -8064.553} C_VEL
LIN {X 0,Y 460.503,Z 200.422,A -85,B 0,C 180,E1 -8067.714,E2 -8067.714} C_VEL
LIN {X 0,Y 460.51,Z 200.437,A -85,B 0,C 180,E1 -8070.767,E2 -8070.767} C_VEL
LIN {X 0,Y 460.532,Z 200.417,A -85,B 0,C 180,E1 -8073.733,E2 -8073.733} C_VEL
LIN {X 0,Y 460.52,Z 200.434,A -85,B 0,C 180,E1 -8076.623,E2 -8076.623} C_VEL
LIN {X 0,Y 460.541,Z 200.416,A -85,B 0,C 180,E1 -8079.453,E2 -8079.453} C_VEL
LIN {X 0,Y 460.526,Z 200.425,A -85,B 0,C 180,E1 -8082.229,E2 -8082.229} C_VEL
LIN {X 0,Y 460.532,Z 200.429,A -85,B 0,C 180,E1 -8084.964,E2 -8084.964} C_VEL
LIN {X 0,Y 460.597,Z 200.399,A -85,B 0,C 180,E1 -8087.666,E2 -8087.666} C_VEL
LIN {X 0,Y 460.597,Z 200.423,A -85,B 0,C 180,E1 -8091.224,E2 -8091.224} C_VEL
LIN {X 0,Y 460.683,Z 200.405,A -85,B 0,C 180,E1 -8093.87,E2 -8093.87} C_VEL
LIN {X 0,Y 460.791,Z 200.384,A -85,B 0,C 180,E1 -8097.378,E2 -8097.378} C_VEL
LIN {X 0,Y 460.818,Z 200.391,A -85,B 0,C 180,E1 -8100,E2 -8100} C_VEL
LIN {X 0,Y 460.791,Z 200.397,A -85,B 0,C 180,E1 -8102.623,E2 -8102.623} C_VEL
LIN {X 0,Y 460.679,Z 200.404,A -85,B 0,C 180,E1 -8106.131,E2 -8106.131} C_VEL
LIN {X 0,Y 460.597,Z 200.423,A -85,B 0,C 180,E1 -8108.777,E2 -8108.777} C_VEL
LIN {X 0,Y 460.582,Z 200.413,A -85,B 0,C 180,E1 -8112.446,E2 -8112.446} C_VEL
LIN {X 0,Y 460.591,Z 200.421,A -85,B 0,C 180,E1 -8116.009,E2 -8116.009} C_VEL
LIN {X 0,Y 460.54,Z 200.416,A -85,B 0,C 180,E1 -8119.617,E2 -8119.617} C_VEL
LIN {X 0,Y 460.487,Z 200.44,A -85,B 0,C 180,E1 -8122.43,E2 -8122.43} C_VEL
LIN {X 0,Y 460.54,Z 200.418,A -85,B 0,C 180,E1 -8125.804,E2 -8125.804} C_VEL
LIN {X 0,Y 460.526,Z 200.43,A -85,B 0,C 180,E1 -8128.235,E2 -8128.235} C_VEL
LIN {X 0,Y 460.494,Z 200.429,A -85,B 0,C 180,E1 -8131.285,E2 -8131.285} C_VEL
LIN {X 0,Y 460.51,Z 200.433,A -85,B 0,C 180,E1 -8134.508,E2 -8134.508} C_VEL
LIN {X 0,Y 460.479,Z 200.434,A -85,B 0,C 180,E1 -8137.626,E2 -8137.626} C_VEL
LIN {X 0,Y 460.518,Z 200.427,A -85,B 0,C 180,E1 -8140.272,E2 -8140.272} C_VEL
LIN {X 0,Y 460.477,Z 200.434,A -85,B 0,C 180,E1 -8143.379,E2 -8143.379} C_VEL
LIN {X 0,Y 460.491,Z 200.436,A -85,B 0,C 180,E1 -8146.629,E2 -8146.629} C_VEL
LIN {X 0,Y 460.519,Z 200.431,A -85,B 0,C 180,E1 -8149.735,E2 -8149.735} C_VEL
LIN {X 0,Y 460.513,Z 200.434,A -85,B 0,C 180,E1 -8152.523,E2 -8152.523} C_VEL
LIN {X 0,Y 460.536,Z 200.423,A -85,B 0,C 180,E1 -8155.627,E2 -8155.627} C_VEL
LIN {X 0,Y 460.528,Z 200.428,A -85,B 0,C 180,E1 -8158.748,E2 -8158.748} C_VEL
LIN {X 0,Y 460.543,Z 200.432,A -85,B 0,C 180,E1 -8162.264,E2 -8162.264} C_VEL
LIN {X 0,Y 460.526,Z 200.429,A -85,B 0,C 180,E1 -8164.707,E2 -8164.707} C_VEL
LIN {X 0,Y 460.505,Z 200.432,A -85,B 0,C 180,E1 -8167.574,E2 -8167.574} C_VEL
LIN {X 0,Y 460.561,Z 200.425,A -85,B 0,C 180,E1 -8170.387,E2 -8170.387} C_VEL
LIN {X 0,Y 460.565,Z 200.429,A -85,B 0,C 180,E1 -8174.06,E2 -8174.06} C_VEL
LIN {X 0,Y 460.61,Z 200.424,A -85,B 0,C 180,E1 -8177.669,E2 -8177.669} C_VEL
LIN {X 0,Y 460.571,Z 200.426,A -85,B 0,C 180,E1 -8179.261,E2 -8179.261} C_VEL
LIN {X 0,Y 459.91,Z 200.513,A -85,B 0,C 180,E1 -8179.991,E2 -8179.991} C_VEL
LIN {X 0,Y 457.069,Z 200.871,A -85,B 0,C 180,E1 -8181.177,E2 -8181.177} C_VEL
LIN {X 0,Y 454.675,Z 201.167,A -85,B 0,C 180,E1 -8182.133,E2 -8182.133} C_VEL
LIN {X 0,Y 453.663,Z 201.288,A -85,B 0,C 180,E1 -8182.872,E2 -8182.872} C_VEL
LIN {X 0,Y 453.589,Z 201.294,A -85,B 0,C 180,E1 -8183.122,E2 -8183.122} C_VEL
LIN {X 0,Y 453.509,Z 201.3,A -85,B 0,C 180,E1 -8185.336,E2 -8185.336} C_VEL
LIN {X 0,Y 453.515,Z 201.372,A -85,B 0,C 180,E1 -8185.503,E2 -8185.503} C_VEL
LIN {X 0,Y 455.942,Z 209.164,A -85,B 0,C 180,E1 -8186.704,E2 -8186.704} C_VEL
LIN {X 0,Y 463.11,Z 224.053,A -85,B 0,C 180,E1 -8187.478,E2 -8187.478} C_VEL
LIN {X 0,Y 467.624,Z 233.876,A -85,B 0,C 180,E1 -8187.96,E2 -8187.96} C_VEL
LIN {X 0,Y 464.663,Z 414.878,A -85,B 0,C 180,E1 -8190.924,E2 -8190.924} C_VEL
LIN {X 0,Y 464.006,Z 431.727,A -85,B 0,C 180,E1 -8191.373,E2 -8191.373} C_VEL
LIN {X 0,Y 463.285,Z 447.22,A -85,B 0,C 180,E1 -8191.958,E2 -8191.958} C_VEL
LIN {X 0,Y 462.417,Z 461.051,A -85,B 0,C 180,E1 -8192.615,E2 -8192.615} C_VEL
LIN {X 0,Y 461.359,Z 475.824,A -85,B 0,C 180,E1 -8193.495,E2 -8193.495} C_VEL
LIN {X 0,Y 460.226,Z 489.628,A -85,B 0,C 180,E1 -8194.491,E2 -8194.491} C_VEL
LIN {X 0,Y 459.041,Z 502.985,A -85,B 0,C 180,E1 -8195.633,E2 -8195.633} C_VEL
LIN {X 0,Y 457.909,Z 515.921,A -85,B 0,C 180,E1 -8196.944,E2 -8196.944} C_VEL
LIN {X 0,Y 456.708,Z 528.124,A -85,B 0,C 180,E1 -8198.408,E2 -8198.408} C_VEL
LIN {X 0,Y 455.631,Z 539.373,A -85,B 0,C 180,E1 -8199.995,E2 -8199.995} C_VEL
LIN {X 0,Y 454.669,Z 550.284,A -85,B 0,C 180,E1 -8201.82,E2 -8201.82} C_VEL
LIN {X 0,Y 453.951,Z 559.477,A -85,B 0,C 180,E1 -8203.658,E2 -8203.658} C_VEL
LIN {X 0,Y 453.363,Z 567.65,A -85,B 0,C 180,E1 -8205.63,E2 -8205.63} C_VEL
LIN {X 0,Y 452.935,Z 574.297,A -85,B 0,C 180,E1 -8207.614,E2 -8207.614} C_VEL
LIN {X 0,Y 452.724,Z 579.26,A -85,B 0,C 180,E1 -8209.499,E2 -8209.499} C_VEL
LIN {X 0,Y 452.481,Z 582.905,A -85,B 0,C 180,E1 -8211.261,E2 -8211.261} C_VEL
LIN {X 0,Y 452.323,Z 586.13,A -85,B 0,C 180,E1 -8213.548,E2 -8213.548} C_VEL
LIN {X 0,Y 452.269,Z 587.738,A -85,B 0,C 180,E1 -8215.793,E2 -8215.793} C_VEL
LIN {X 0,Y 452.304,Z 587.862,A -85,B 0,C 180,E1 -8217.786,E2 -8217.786} C_VEL
LIN {X 0,Y 452.357,Z 586.816,A -85,B 0,C 180,E1 -8219.814,E2 -8219.814} C_VEL
LIN {X 0,Y 452.432,Z 584.501,A -85,B 0,C 180,E1 -8221.882,E2 -8221.882} C_VEL
LIN {X 0,Y 452.624,Z 580.737,A -85,B 0,C 180,E1 -8223.986,E2 -8223.986} C_VEL
LIN {X 0,Y 452.925,Z 575.195,A -85,B 0,C 180,E1 -8226.207,E2 -8226.207} C_VEL
LIN {X 0,Y 453.332,Z 568.293,A -85,B 0,C 180,E1 -8228.326,E2 -8228.326} C_VEL
LIN {X 0,Y 453.914,Z 560.394,A -85,B 0,C 180,E1 -8230.273,E2 -8230.273} C_VEL
LIN {X 0,Y 454.617,Z 551.5,A -85,B 0,C 180,E1 -8232.094,E2 -8232.094} C_VEL
LIN {X 0,Y 455.474,Z 542.371,A -85,B 0,C 180,E1 -8233.683,E2 -8233.683} C_VEL
LIN {X 0,Y 456.546,Z 530.705,A -85,B 0,C 180,E1 -8235.396,E2 -8235.396} C_VEL
LIN {X 0,Y 457.683,Z 519.081,A -85,B 0,C 180,E1 -8236.836,E2 -8236.836} C_VEL
LIN {X 0,Y 458.854,Z 506.612,A -85,B 0,C 180,E1 -8238.16,E2 -8238.16} C_VEL
LIN {X 0,Y 460.09,Z 493.087,A -85,B 0,C 180,E1 -8239.378,E2 -8239.378} C_VEL
LIN {X 0,Y 461.338,Z 478.269,A -85,B 0,C 180,E1 -8240.488,E2 -8240.488} C_VEL
LIN {X 0,Y 462.494,Z 462.255,A -85,B 0,C 180,E1 -8241.462,E2 -8241.462} C_VEL
LIN {X 0,Y 463.447,Z 447.057,A -85,B 0,C 180,E1 -8242.192,E2 -8242.192} C_VEL
LIN {X 0,Y 464.261,Z 430.585,A -85,B 0,C 180,E1 -8242.8,E2 -8242.8} C_VEL
LIN {X 0,Y 464.863,Z 414.08,A -85,B 0,C 180,E1 -8243.227,E2 -8243.227} C_VEL
LIN {X 0,Y 468.001,Z 234.683,A -85,B 0,C 180,E1 -8246.18,E2 -8246.18} C_VEL
LIN {X 0,Y 464.451,Z 226.557,A -85,B 0,C 180,E1 -8246.581,E2 -8246.581} C_VEL
LIN {X 0,Y 456.131,Z 209.871,A -85,B 0,C 180,E1 -8247.509,E2 -8247.509} C_VEL
LIN {X 0,Y 453.503,Z 201.31,A -85,B 0,C 180,E1 -8248.898,E2 -8248.898} C_VEL
LIN {X 0,Y 453.539,Z 201.304,A -85,B 0,C 180,E1 -8252.297,E2 -8252.297} C_VEL
LIN {X 0,Y 453.503,Z 201.31,A -85,B 0,C 180,E1 -8255.264,E2 -8255.264} C_VEL
LIN {X 0,Y 453.482,Z 201.308,A -85,B 0,C 180,E1 -8258.415,E2 -8258.415} C_VEL
LIN {X 0,Y 453.524,Z 201.304,A -85,B 0,C 180,E1 -8261.008,E2 -8261.008} C_VEL
LIN {X 0,Y 453.57,Z 201.299,A -85,B 0,C 180,E1 -8263.879,E2 -8263.879} C_VEL
LIN {X 0,Y 453.565,Z 201.298,A -85,B 0,C 180,E1 -8267.471,E2 -8267.471} C_VEL
LIN {X 0,Y 453.59,Z 201.295,A -85,B 0,C 180,E1 -8271.086,E2 -8271.086} C_VEL
LIN {X 0,Y 453.675,Z 201.286,A -85,B 0,C 180,E1 -8273.774,E2 -8273.774} C_VEL
LIN {X 0,Y 453.741,Z 201.276,A -85,B 0,C 180,E1 -8277.336,E2 -8277.336} C_VEL
LIN {X 0,Y 453.82,Z 201.269,A -85,B 0,C 180,E1 -8280,E2 -8280} C_VEL
LIN {X 0,Y 453.741,Z 201.275,A -85,B 0,C 180,E1 -8282.663,E2 -8282.663} C_VEL
LIN {X 0,Y 453.664,Z 201.285,A -85,B 0,C 180,E1 -8286.225,E2 -8286.225} C_VEL
LIN {X 0,Y 453.584,Z 201.295,A -85,B 0,C 180,E1 -8288.913,E2 -8288.913} C_VEL
LIN {X 0,Y 453.563,Z 201.296,A -85,B 0,C 180,E1 -8292.528,E2 -8292.528} C_VEL
LIN {X 0,Y 453.544,Z 201.298,A -85,B 0,C 180,E1 -8296.196,E2 -8296.196} C_VEL
LIN {X 0,Y 453.516,Z 201.304,A -85,B 0,C 180,E1 -8299.039,E2 -8299.039} C_VEL
LIN {X 0,Y 453.475,Z 201.309,A -85,B 0,C 180,E1 -8301.836,E2 -8301.836} C_VEL
LIN {X 0,Y 453.499,Z 201.303,A -85,B 0,C 180,E1 -8304.735,E2 -8304.735} C_VEL
LIN {X 0,Y 453.531,Z 201.302,A -85,B 0,C 180,E1 -8307.959,E2 -8307.959} C_VEL
LIN {X 0,Y 453.463,Z 201.31,A -85,B 0,C 180,E1 -8311.524,E2 -8311.524} C_VEL
LIN {X 0,Y 453.482,Z 201.308,A -85,B 0,C 180,E1 -8314.776,E2 -8314.776} C_VEL
LIN {X 0,Y 453.461,Z 201.31,A -85,B 0,C 180,E1 -8318.311,E2 -8318.311} C_VEL
LIN {X 0,Y 453.494,Z 201.306,A -85,B 0,C 180,E1 -8320.608,E2 -8320.608} C_VEL
LIN {X 0,Y 453.46,Z 201.311,A -85,B 0,C 180,E1 -8324.221,E2 -8324.221} C_VEL
LIN {X 0,Y 453.437,Z 201.315,A -85,B 0,C 180,E1 -8327.001,E2 -8327.001} C_VEL
LIN {X 0,Y 453.472,Z 201.312,A -85,B 0,C 180,E1 -8329.412,E2 -8329.412} C_VEL
LIN {X 0,Y 453.45,Z 201.312,A -85,B 0,C 180,E1 -8332.809,E2 -8332.809} C_VEL
LIN {X 0,Y 453.535,Z 201.365,A -85,B 0,C 180,E1 -8335.756,E2 -8335.756} C_VEL
LIN {X 0,Y 459.695,Z 220.707,A -85,B 0,C 180,E1 -8338.568,E2 -8338.568} C_VEL
LIN {X 0,Y 462.73,Z 231.628,A -85,B 0,C 180,E1 -8340.024,E2 -8340.024} C_VEL
LIN {X 0,Y 467.682,Z 260.117,A -85,B 0,C 180,E1 -8340.888,E2 -8340.888} C_VEL
LIN {X 0,Y 464.595,Z 439.135,A -85,B 0,C 180,E1 -8343.83,E2 -8343.83} C_VEL
LIN {X 0,Y 463.838,Z 455.652,A -85,B 0,C 180,E1 -8344.265,E2 -8344.265} C_VEL
LIN {X 0,Y 462.973,Z 471.299,A -85,B 0,C 180,E1 -8344.845,E2 -8344.845} C_VEL
LIN {X 0,Y 461.878,Z 487.387,A -85,B 0,C 180,E1 -8345.622,E2 -8345.622} C_VEL
LIN {X 0,Y 460.799,Z 502.33,A -85,B 0,C 180,E1 -8346.527,E2 -8346.527} C_VEL
LIN {X 0,Y 459.523,Z 515.874,A -85,B 0,C 180,E1 -8347.519,E2 -8347.519} C_VEL
LIN {X 0,Y 458.248,Z 530.003,A -85,B 0,C 180,E1 -8348.755,E2 -8348.755} C_VEL
LIN {X 0,Y 457.11,Z 542.715,A -85,B 0,C 180,E1 -8350.071,E2 -8350.071} C_VEL
LIN {X 0,Y 455.953,Z 555.141,A -85,B 0,C 180,E1 -8351.578,E2 -8351.578} C_VEL
LIN {X 0,Y 454.92,Z 567.085,A -85,B 0,C 180,E1 -8353.3,E2 -8353.3} C_VEL
LIN {X 0,Y 454.127,Z 576.872,A -85,B 0,C 180,E1 -8354.975,E2 -8354.975} C_VEL
LIN {X 0,Y 453.507,Z 585.854,A -85,B 0,C 180,E1 -8356.785,E2 -8356.785} C_VEL
LIN {X 0,Y 453.139,Z 592.541,A -85,B 0,C 180,E1 -8358.366,E2 -8358.366} C_VEL
LIN {X 0,Y 452.713,Z 600.286,A -85,B 0,C 180,E1 -8360.617,E2 -8360.617} C_VEL
LIN {X 0,Y 452.57,Z 606.182,A -85,B 0,C 180,E1 -8362.862,E2 -8362.862} C_VEL
LIN {X 0,Y 452.496,Z 609.635,A -85,B 0,C 180,E1 -8364.651,E2 -8364.651} C_VEL
LIN {X 0,Y 452.428,Z 612.144,A -85,B 0,C 180,E1 -8366.436,E2 -8366.436} C_VEL
LIN {X 0,Y 452.451,Z 613.566,A -85,B 0,C 180,E1 -8368.218,E2 -8368.218} C_VEL
LIN {X 0,Y 452.43,Z 614.106,A -85,B 0,C 180,E1 -8369.998,E2 -8369.998} C_VEL
LIN {X 0,Y 452.45,Z 613.583,A -85,B 0,C 180,E1 -8371.778,E2 -8371.778} C_VEL
LIN {X 0,Y 452.427,Z 612.178,A -85,B 0,C 180,E1 -8373.56,E2 -8373.56} C_VEL
LIN {X 0,Y 452.494,Z 609.688,A -85,B 0,C 180,E1 -8375.345,E2 -8375.345} C_VEL
LIN {X 0,Y 452.566,Z 606.254,A -85,B 0,C 180,E1 -8377.134,E2 -8377.134} C_VEL
LIN {X 0,Y 452.718,Z 600.38,A -85,B 0,C 180,E1 -8379.379,E2 -8379.379} C_VEL
LIN {X 0,Y 453.139,Z 592.65,A -85,B 0,C 180,E1 -8381.629,E2 -8381.629} C_VEL
LIN {X 0,Y 453.653,Z 583.932,A -85,B 0,C 180,E1 -8383.663,E2 -8383.663} C_VEL
LIN {X 0,Y 454.407,Z 574.515,A -85,B 0,C 180,E1 -8385.471,E2 -8385.471} C_VEL
LIN {X 0,Y 455.134,Z 564.806,A -85,B 0,C 180,E1 -8387.058,E2 -8387.058} C_VEL
LIN {X 0,Y 456.147,Z 553.492,A -85,B 0,C 180,E1 -8388.642,E2 -8388.642} C_VEL
LIN {X 0,Y 457.232,Z 541.489,A -85,B 0,C 180,E1 -8390.078,E2 -8390.078} C_VEL
LIN {X 0,Y 458.485,Z 527.709,A -85,B 0,C 180,E1 -8391.464,E2 -8391.464} C_VEL
LIN {X 0,Y 459.667,Z 514.445,A -85,B 0,C 180,E1 -8392.587,E2 -8392.587} C_VEL
LIN {X 0,Y 460.929,Z 499.585,A -85,B 0,C 180,E1 -8393.641,E2 -8393.641} C_VEL
LIN {X 0,Y 462.058,Z 484.062,A -85,B 0,C 180,E1 -8394.543,E2 -8394.543} C_VEL
LIN {X 0,Y 463.115,Z 468.285,A -85,B 0,C 180,E1 -8395.262,E2 -8395.262} C_VEL
LIN {X 0,Y 463.908,Z 452.114,A -85,B 0,C 180,E1 -8395.817,E2 -8395.817} C_VEL
LIN {X 0,Y 464.581,Z 435.294,A -85,B 0,C 180,E1 -8396.211,E2 -8396.211} C_VEL
LIN {X 0,Y 467.415,Z 259.389,A -85,B 0,C 180,E1 -8399.079,E2 -8399.079} C_VEL
LIN {X 0,Y 462.643,Z 231.784,A -85,B 0,C 180,E1 -8399.913,E2 -8399.913} C_VEL
LIN {X 0,Y 458.603,Z 217.508,A -85,B 0,C 180,E1 -8401.827,E2 -8401.827} C_VEL
LIN {X 0,Y 453.501,Z 201.306,A -85,B 0,C 180,E1 -8404.141,E2 -8404.141} C_VEL
LIN {X 0,Y 453.43,Z 201.315,A -85,B 0,C 180,E1 -8407.77,E2 -8407.77} C_VEL
LIN {X 0,Y 453.473,Z 201.307,A -85,B 0,C 180,E1 -8410.606,E2 -8410.606} C_VEL
LIN {X 0,Y 453.434,Z 201.314,A -85,B 0,C 180,E1 -8413.242,E2 -8413.242} C_VEL
LIN {X 0,Y 453.451,Z 201.308,A -85,B 0,C 180,E1 -8415.778,E2 -8415.778} C_VEL
LIN {X 0,Y 453.492,Z 201.304,A -85,B 0,C 180,E1 -8419.404,E2 -8419.404} C_VEL
LIN {X 0,Y 453.449,Z 201.311,A -85,B 0,C 180,E1 -8422.221,E2 -8422.221} C_VEL
LIN {X 0,Y 453.462,Z 201.315,A -85,B 0,C 180,E1 -8425.221,E2 -8425.221} C_VEL
LIN {X 0,Y 453.437,Z 201.303,A -85,B 0,C 180,E1 -8428.473,E2 -8428.473} C_VEL
LIN {X 0,Y 453.502,Z 201.303,A -85,B 0,C 180,E1 -8432.039,E2 -8432.039} C_VEL
LIN {X 0,Y 453.485,Z 201.309,A -85,B 0,C 180,E1 -8435.264,E2 -8435.264} C_VEL
LIN {X 0,Y 453.505,Z 201.305,A -85,B 0,C 180,E1 -8438.396,E2 -8438.396} C_VEL
LIN {X 0,Y 453.49,Z 201.297,A -85,B 0,C 180,E1 -8441.008,E2 -8441.008} C_VEL
LIN {X 0,Y 453.536,Z 201.3,A -85,B 0,C 180,E1 -8443.879,E2 -8443.879} C_VEL
LIN {X 0,Y 453.569,Z 201.274,A -85,B 0,C 180,E1 -8447.472,E2 -8447.472} C_VEL
LIN {X 0,Y 453.561,Z 201.301,A -85,B 0,C 180,E1 -8451.086,E2 -8451.086} C_VEL
LIN {X 0,Y 453.649,Z 201.281,A -85,B 0,C 180,E1 -8453.775,E2 -8453.775} C_VEL
LIN {X 0,Y 453.732,Z 201.264,A -85,B 0,C 180,E1 -8457.337,E2 -8457.337} C_VEL
LIN {X 0,Y 453.789,Z 201.267,A -85,B 0,C 180,E1 -8460,E2 -8460} C_VEL
LIN {X 0,Y 453.732,Z 201.275,A -85,B 0,C 180,E1 -8462.664,E2 -8462.664} C_VEL
LIN {X 0,Y 453.646,Z 201.281,A -85,B 0,C 180,E1 -8466.226,E2 -8466.226} C_VEL
LIN {X 0,Y 453.561,Z 201.297,A -85,B 0,C 180,E1 -8468.914,E2 -8468.914} C_VEL
LIN {X 0,Y 453.532,Z 201.292,A -85,B 0,C 180,E1 -8472.53,E2 -8472.53} C_VEL
LIN {X 0,Y 453.526,Z 201.303,A -85,B 0,C 180,E1 -8476.197,E2 -8476.197} C_VEL
LIN {X 0,Y 453.49,Z 201.296,A -85,B 0,C 180,E1 -8479.042,E2 -8479.042} C_VEL
LIN {X 0,Y 453.45,Z 201.31,A -85,B 0,C 180,E1 -8481.838,E2 -8481.838} C_VEL
LIN {X 0,Y 453.487,Z 201.299,A -85,B 0,C 180,E1 -8484.737,E2 -8484.737} C_VEL
LIN {X 0,Y 453.505,Z 201.301,A -85,B 0,C 180,E1 -8487.962,E2 -8487.962} C_VEL
LIN {X 0,Y 453.44,Z 201.308,A -85,B 0,C 180,E1 -8491.527,E2 -8491.527} C_VEL
LIN {X 0,Y 453.465,Z 201.31,A -85,B 0,C 180,E1 -8494.78,E2 -8494.78} C_VEL
LIN {X 0,Y 453.438,Z 201.308,A -85,B 0,C 180,E1 -8498.315,E2 -8498.315} C_VEL
LIN {X 0,Y 453.474,Z 201.31,A -85,B 0,C 180,E1 -8500.612,E2 -8500.612} C_VEL
LIN {X 0,Y 453.433,Z 201.312,A -85,B 0,C 180,E1 -8503.247,E2 -8503.247} C_VEL
LIN {X 0,Y 453.442,Z 201.304,A -85,B 0,C 180,E1 -8505.781,E2 -8505.781} C_VEL
LIN {X 0,Y 453.478,Z 201.305,A -85,B 0,C 180,E1 -8509.412,E2 -8509.412} C_VEL
LIN {X 0,Y 453.457,Z 201.311,A -85,B 0,C 180,E1 -8512.815,E2 -8512.815} C_VEL
LIN {X 0,Y 453.466,Z 201.306,A -85,B 0,C 180,E1 -8516.09,E2 -8516.09} C_VEL
LIN {X 0,Y 453.466,Z 201.307,A -85,B 0,C 180,E1 -8519.244,E2 -8519.244} C_VEL
LIN {X 0,Y 453.499,Z 201.309,A -85,B 0,C 180,E1 -8522.299,E2 -8522.299} C_VEL
LIN {X 0,Y 453.487,Z 201.305,A -85,B 0,C 180,E1 -8525.267,E2 -8525.267} C_VEL
LIN {X 0,Y 453.476,Z 201.311,A -85,B 0,C 180,E1 -8528.418,E2 -8528.418} C_VEL
LIN {X 0,Y 453.52,Z 201.3,A -85,B 0,C 180,E1 -8531.012,E2 -8531.012} C_VEL
LIN {X 0,Y 453.519,Z 201.305,A -85,B 0,C 180,E1 -8534.728,E2 -8534.728} C_VEL
LIN {X 0,Y 453.559,Z 201.299,A -85,B 0,C 180,E1 -8538.382,E2 -8538.382} C_VEL
LIN {X 0,Y 453.578,Z 201.298,A -85,B 0,C 180,E1 -8541.089,E2 -8541.089} C_VEL
LIN {X 0,Y 453.589,Z 201.294,A -85,B 0,C 180,E1 -8543.122,E2 -8543.122} C_VEL
LIN {X 0,Y 452.909,Z 201.377,A -85,B 0,C 180,E1 -8543.641,E2 -8543.641} C_VEL
LIN {X 0,Y 450.095,Z 202.005,A -85,B 0,C 180,E1 -8544.457,E2 -8544.457} C_VEL
LIN {X 0,Y 448.024,Z 203.423,A -85,B 0,C 180,E1 -8545.072,E2 -8545.072} C_VEL
LIN {X 0,Y 447.444,Z 205.258,A -85,B 0,C 180,E1 -8545.514,E2 -8545.514} C_VEL
LIN {X 0,Y 447.581,Z 206.038,A -85,B 0,C 180,E1 -8545.648,E2 -8545.648} C_VEL
LIN {X 0,Y 448.746,Z 209.655,A -85,B 0,C 180,E1 -8546.183,E2 -8546.183} C_VEL
LIN {X 0,Y 454.297,Z 220.599,A -85,B 0,C 180,E1 -8546.794,E2 -8546.794} C_VEL
LIN {X 0,Y 461.392,Z 235.958,A -85,B 0,C 180,E1 -8547.571,E2 -8547.571} C_VEL
LIN {X 0,Y 458.244,Z 415.462,A -85,B 0,C 180,E1 -8550.551,E2 -8550.551} C_VEL
LIN {X 0,Y 457.551,Z 433.017,A -85,B 0,C 180,E1 -8551.033,E2 -8551.033} C_VEL
LIN {X 0,Y 456.686,Z 449.472,A -85,B 0,C 180,E1 -8551.679,E2 -8551.679} C_VEL
LIN {X 0,Y 455.669,Z 464.375,A -85,B 0,C 180,E1 -8552.433,E2 -8552.433} C_VEL
LIN {X 0,Y 454.604,Z 478.684,A -85,B 0,C 180,E1 -8553.326,E2 -8553.326} C_VEL
LIN {X 0,Y 453.293,Z 493.503,A -85,B 0,C 180,E1 -8554.448,E2 -8554.448} C_VEL
LIN {X 0,Y 452.023,Z 507.046,A -85,B 0,C 180,E1 -8555.689,E2 -8555.689} C_VEL
LIN {X 0,Y 450.889,Z 518.698,A -85,B 0,C 180,E1 -8556.94,E2 -8556.94} C_VEL
LIN {X 0,Y 449.764,Z 529.774,A -85,B 0,C 180,E1 -8558.312,E2 -8558.312} C_VEL
LIN {X 0,Y 448.674,Z 540.786,A -85,B 0,C 180,E1 -8559.924,E2 -8559.924} C_VEL
LIN {X 0,Y 447.765,Z 550.264,A -85,B 0,C 180,E1 -8561.546,E2 -8561.546} C_VEL
LIN {X 0,Y 447.036,Z 558.733,A -85,B 0,C 180,E1 -8563.236,E2 -8563.236} C_VEL
LIN {X 0,Y 446.434,Z 566.341,A -85,B 0,C 180,E1 -8565.057,E2 -8565.057} C_VEL
LIN {X 0,Y 445.972,Z 572.892,A -85,B 0,C 180,E1 -8566.952,E2 -8566.952} C_VEL
LIN {X 0,Y 445.705,Z 578.329,A -85,B 0,C 180,E1 -8568.896,E2 -8568.896} C_VEL
LIN {X 0,Y 445.504,Z 581.459,A -85,B 0,C 180,E1 -8570.309,E2 -8570.309} C_VEL
LIN {X 0,Y 445.289,Z 584.829,A -85,B 0,C 180,E1 -8572.26,E2 -8572.26} C_VEL
LIN {X 0,Y 445.19,Z 586.984,A -85,B 0,C 180,E1 -8574.234,E2 -8574.234} C_VEL
LIN {X 0,Y 445.184,Z 588.047,A -85,B 0,C 180,E1 -8576.235,E2 -8576.235} C_VEL
LIN {X 0,Y 445.201,Z 587.982,A -85,B 0,C 180,E1 -8578.268,E2 -8578.268} C_VEL
LIN {X 0,Y 445.272,Z 586.609,A -85,B 0,C 180,E1 -8580.338,E2 -8580.338} C_VEL
LIN {X 0,Y 445.387,Z 583.939,A -85,B 0,C 180,E1 -8582.447,E2 -8582.447} C_VEL
LIN {X 0,Y 445.591,Z 579.839,A -85,B 0,C 180,E1 -8584.598,E2 -8584.598} C_VEL
LIN {X 0,Y 445.894,Z 575.013,A -85,B 0,C 180,E1 -8586.501,E2 -8586.501} C_VEL
LIN {X 0,Y 446.324,Z 568.538,A -85,B 0,C 180,E1 -8588.497,E2 -8588.497} C_VEL
LIN {X 0,Y 446.83,Z 562.035,A -85,B 0,C 180,E1 -8590.157,E2 -8590.157} C_VEL
LIN {X 0,Y 447.505,Z 554.121,A -85,B 0,C 180,E1 -8591.872,E2 -8591.872} C_VEL
LIN {X 0,Y 448.367,Z 544.602,A -85,B 0,C 180,E1 -8593.606,E2 -8593.606} C_VEL
LIN {X 0,Y 449.491,Z 533.744,A -85,B 0,C 180,E1 -8595.283,E2 -8595.283} C_VEL
LIN {X 0,Y 450.71,Z 521.981,A -85,B 0,C 180,E1 -8596.829,E2 -8596.829} C_VEL
LIN {X 0,Y 451.991,Z 509.011,A -85,B 0,C 180,E1 -8598.276,E2 -8598.276} C_VEL
LIN {X 0,Y 453.368,Z 494.799,A -85,B 0,C 180,E1 -8599.599,E2 -8599.599} C_VEL
LIN {X 0,Y 454.709,Z 479.871,A -85,B 0,C 180,E1 -8600.748,E2 -8600.748} C_VEL
LIN {X 0,Y 455.802,Z 465.654,A -85,B 0,C 180,E1 -8601.652,E2 -8601.652} C_VEL
LIN {X 0,Y 456.858,Z 450.301,A -85,B 0,C 180,E1 -8602.441,E2 -8602.441} C_VEL
LIN {X 0,Y 457.767,Z 434.269,A -85,B 0,C 180,E1 -8603.079,E2 -8603.079} C_VEL
LIN {X 0,Y 458.446,Z 417.14,A -85,B 0,C 180,E1 -8603.561,E2 -8603.561} C_VEL
LIN {X 0,Y 459.181,Z 376.829,A -85,B 0,C 180,E1 -8604.261,E2 -8604.261} C_VEL
LIN {X 0,Y 461.785,Z 236.28,A -85,B 0,C 180,E1 -8606.6,E2 -8606.6} C_VEL
LIN {X 0,Y 452.466,Z 216.959,A -85,B 0,C 180,E1 -8607.662,E2 -8607.662} C_VEL
LIN {X 0,Y 448.924,Z 210.046,A -85,B 0,C 180,E1 -8608.086,E2 -8608.086} C_VEL
LIN {X 0,Y 446.431,Z 202.187,A -85,B 0,C 180,E1 -8609.39,E2 -8609.39} C_VEL
LIN {X 0,Y 446.475,Z 202.184,A -85,B 0,C 180,E1 -8612.838,E2 -8612.838} C_VEL
LIN {X 0,Y 446.465,Z 202.183,A -85,B 0,C 180,E1 -8615.924,E2 -8615.924} C_VEL
LIN {X 0,Y 446.455,Z 202.18,A -85,B 0,C 180,E1 -8618.773,E2 -8618.773} C_VEL
LIN {X 0,Y 446.459,Z 202.184,A -85,B 0,C 180,E1 -8621.649,E2 -8621.649} C_VEL
LIN {X 0,Y 446.509,Z 202.178,A -85,B 0,C 180,E1 -8624.479,E2 -8624.479} C_VEL
LIN {X 0,Y 446.517,Z 202.179,A -85,B 0,C 180,E1 -8628.193,E2 -8628.193} C_VEL
LIN {X 0,Y 446.601,Z 202.167,A -85,B 0,C 180,E1 -8631.857,E2 -8631.857} C_VEL
LIN {X 0,Y 446.643,Z 202.16,A -85,B 0,C 180,E1 -8634.582,E2 -8634.582} C_VEL
LIN {X 0,Y 446.661,Z 202.157,A -85,B 0,C 180,E1 -8638.196,E2 -8638.196} C_VEL
LIN {X 0,Y 446.79,Z 202.145,A -85,B 0,C 180,E1 -8640,E2 -8640} C_VEL
LIN {X 0,Y 446.688,Z 202.153,A -85,B 0,C 180,E1 -8642.705,E2 -8642.705} C_VEL
LIN {X 0,Y 446.632,Z 202.161,A -85,B 0,C 180,E1 -8646.323,E2 -8646.323} C_VEL
LIN {X 0,Y 446.532,Z 202.175,A -85,B 0,C 180,E1 -8649.055,E2 -8649.055} C_VEL
LIN {X 0,Y 446.521,Z 202.174,A -85,B 0,C 180,E1 -8652.729,E2 -8652.729} C_VEL
LIN {X 0,Y 446.488,Z 202.176,A -85,B 0,C 180,E1 -8656.459,E2 -8656.459} C_VEL
LIN {X 0,Y 446.467,Z 202.182,A -85,B 0,C 180,E1 -8659.303,E2 -8659.303} C_VEL
LIN {X 0,Y 446.416,Z 202.186,A -85,B 0,C 180,E1 -8662.199,E2 -8662.199} C_VEL
LIN {X 0,Y 446.442,Z 202.185,A -85,B 0,C 180,E1 -8665.153,E2 -8665.153} C_VEL
LIN {X 0,Y 446.485,Z 202.179,A -85,B 0,C 180,E1 -8668.178,E2 -8668.178} C_VEL
LIN {X 0,Y 446.415,Z 202.187,A -85,B 0,C 180,E1 -8671.773,E2 -8671.773} C_VEL
LIN {X 0,Y 446.422,Z 202.186,A -85,B 0,C 180,E1 -8674.523,E2 -8674.523} C_VEL
LIN {X 0,Y 446.414,Z 202.188,A -85,B 0,C 180,E1 -8678.078,E2 -8678.078} C_VEL
LIN {X 0,Y 446.422,Z 202.184,A -85,B 0,C 180,E1 -8680.916,E2 -8680.916} C_VEL
LIN {X 0,Y 446.398,Z 202.19,A -85,B 0,C 180,E1 -8683.846,E2 -8683.846} C_VEL
LIN {X 0,Y 446.393,Z 202.197,A -85,B 0,C 180,E1 -8686.404,E2 -8686.404} C_VEL
LIN {X 0,Y 446.403,Z 202.191,A -85,B 0,C 180,E1 -8689.797,E2 -8689.797} C_VEL
LIN {X 0,Y 446.406,Z 202.191,A -85,B 0,C 180,E1 -8692.12,E2 -8692.12} C_VEL
LIN {X 0,Y 446.469,Z 202.28,A -85,B 0,C 180,E1 -8695.254,E2 -8695.254} C_VEL
LIN {X 0,Y 452.726,Z 221.581,A -85,B 0,C 180,E1 -8698.141,E2 -8698.141} C_VEL
LIN {X 0,Y 455.488,Z 231.239,A -85,B 0,C 180,E1 -8699.478,E2 -8699.478} C_VEL
LIN {X 0,Y 457.156,Z 235.642,A -85,B 0,C 180,E1 -8699.685,E2 -8699.685} C_VEL
LIN {X 0,Y 461.476,Z 260.648,A -85,B 0,C 180,E1 -8700.458,E2 -8700.458} C_VEL
LIN {X 0,Y 458.265,Z 438.163,A -85,B 0,C 180,E1 -8703.42,E2 -8703.42} C_VEL
LIN {X 0,Y 457.504,Z 454.638,A -85,B 0,C 180,E1 -8703.851,E2 -8703.851} C_VEL
LIN {X 0,Y 456.549,Z 471.16,A -85,B 0,C 180,E1 -8704.466,E2 -8704.466} C_VEL
LIN {X 0,Y 455.366,Z 487.227,A -85,B 0,C 180,E1 -8705.25,E2 -8705.25} C_VEL
LIN {X 0,Y 454.196,Z 502.591,A -85,B 0,C 180,E1 -8706.198,E2 -8706.198} C_VEL
LIN {X 0,Y 452.916,Z 515.698,A -85,B 0,C 180,E1 -8707.173,E2 -8707.173} C_VEL
LIN {X 0,Y 451.667,Z 528.629,A -85,B 0,C 180,E1 -8708.311,E2 -8708.311} C_VEL
LIN {X 0,Y 450.432,Z 541.575,A -85,B 0,C 180,E1 -8709.649,E2 -8709.649} C_VEL
LIN {X 0,Y 449.299,Z 553.168,A -85,B 0,C 180,E1 -8711.059,E2 -8711.059} C_VEL
LIN {X 0,Y 448.229,Z 564.466,A -85,B 0,C 180,E1 -8712.666,E2 -8712.666} C_VEL
LIN {X 0,Y 447.323,Z 575.415,A -85,B 0,C 180,E1 -8714.507,E2 -8714.507} C_VEL
LIN {X 0,Y 446.569,Z 584.62,A -85,B 0,C 180,E1 -8716.344,E2 -8716.344} C_VEL
LIN {X 0,Y 446.116,Z 592.331,A -85,B 0,C 180,E1 -8718.181,E2 -8718.181} C_VEL
LIN {X 0,Y 445.631,Z 600.077,A -85,B 0,C 180,E1 -8720.466,E2 -8720.466} C_VEL
LIN {X 0,Y 445.486,Z 605.974,A -85,B 0,C 180,E1 -8722.748,E2 -8722.748} C_VEL
LIN {X 0,Y 445.399,Z 609.428,A -85,B 0,C 180,E1 -8724.565,E2 -8724.565} C_VEL
LIN {X 0,Y 445.327,Z 611.938,A -85,B 0,C 180,E1 -8726.379,E2 -8726.379} C_VEL
LIN {X 0,Y 445.369,Z 613.361,A -85,B 0,C 180,E1 -8728.189,E2 -8728.189} C_VEL
LIN {X 0,Y 445.337,Z 613.901,A -85,B 0,C 180,E1 -8729.998,E2 -8729.998} C_VEL
LIN {X 0,Y 445.368,Z 613.378,A -85,B 0,C 180,E1 -8731.806,E2 -8731.806} C_VEL
LIN {X 0,Y 445.326,Z 611.971,A -85,B 0,C 180,E1 -8733.617,E2 -8733.617} C_VEL
LIN {X 0,Y 445.397,Z 609.478,A -85,B 0,C 180,E1 -8735.43,E2 -8735.43} C_VEL
LIN {X 0,Y 445.482,Z 606.042,A -85,B 0,C 180,E1 -8737.248,E2 -8737.248} C_VEL
LIN {X 0,Y 445.634,Z 600.161,A -85,B 0,C 180,E1 -8739.529,E2 -8739.529} C_VEL
LIN {X 0,Y 446.113,Z 592.423,A -85,B 0,C 180,E1 -8741.815,E2 -8741.815} C_VEL
LIN {X 0,Y 446.638,Z 583.696,A -85,B 0,C 180,E1 -8743.882,E2 -8743.882} C_VEL
LIN {X 0,Y 447.469,Z 574.272,A -85,B 0,C 180,E1 -8745.717,E2 -8745.717} C_VEL
LIN {X 0,Y 448.237,Z 564.553,A -85,B 0,C 180,E1 -8747.329,E2 -8747.329} C_VEL
LIN {X 0,Y 449.319,Z 553.224,A -85,B 0,C 180,E1 -8748.936,E2 -8748.936} C_VEL
LIN {X 0,Y 450.419,Z 541.614,A -85,B 0,C 180,E1 -8750.346,E2 -8750.346} C_VEL
LIN {X 0,Y 451.663,Z 528.586,A -85,B 0,C 180,E1 -8751.685,E2 -8751.685} C_VEL
LIN {X 0,Y 452.911,Z 515.552,A -85,B 0,C 180,E1 -8752.823,E2 -8752.823} C_VEL
LIN {X 0,Y 454.207,Z 501.428,A -85,B 0,C 180,E1 -8753.863,E2 -8753.863} C_VEL
LIN {X 0,Y 455.422,Z 485.813,A -85,B 0,C 180,E1 -8754.803,E2 -8754.803} C_VEL
LIN {X 0,Y 456.48,Z 470.452,A -85,B 0,C 180,E1 -8755.533,E2 -8755.533} C_VEL
LIN {X 0,Y 457.332,Z 454.312,A -85,B 0,C 180,E1 -8756.124,E2 -8756.124} C_VEL
LIN {X 0,Y 458.1,Z 438.398,A -85,B 0,C 180,E1 -8756.531,E2 -8756.531} C_VEL
LIN {X 0,Y 461.178,Z 260.424,A -85,B 0,C 180,E1 -8759.479,E2 -8759.479} C_VEL
LIN {X 0,Y 456.408,Z 233.928,A -85,B 0,C 180,E1 -8760.287,E2 -8760.287} C_VEL
LIN {X 0,Y 455.497,Z 231.554,A -85,B 0,C 180,E1 -8760.423,E2 -8760.423} C_VEL
LIN {X 0,Y 450.128,Z 213.661,A -85,B 0,C 180,E1 -8762.91,E2 -8762.91} C_VEL
LIN {X 0,Y 446.454,Z 202.189,A -85,B 0,C 180,E1 -8764.616,E2 -8764.616} C_VEL
LIN {X 0,Y 446.395,Z 202.193,A -85,B 0,C 180,E1 -8768.077,E2 -8768.077} C_VEL
LIN {X 0,Y 446.406,Z 202.191,A -85,B 0,C 180,E1 -8770.915,E2 -8770.915} C_VEL
LIN {X 0,Y 446.379,Z 202.194,A -85,B 0,C 180,E1 -8773.843,E2 -8773.843} C_VEL
LIN {X 0,Y 446.398,Z 202.187,A -85,B 0,C 180,E1 -8776.398,E2 -8776.398} C_VEL
LIN {X 0,Y 446.443,Z 202.183,A -85,B 0,C 180,E1 -8779.803,E2 -8779.803} C_VEL
LIN {X 0,Y 446.406,Z 202.188,A -85,B 0,C 180,E1 -8782.121,E2 -8782.121} C_VEL
LIN {X 0,Y 446.403,Z 202.192,A -85,B 0,C 180,E1 -8785.475,E2 -8785.475} C_VEL
LIN {X 0,Y 446.387,Z 202.182,A -85,B 0,C 180,E1 -8788.698,E2 -8788.698} C_VEL
LIN {X 0,Y 446.455,Z 202.181,A -85,B 0,C 180,E1 -8791.82,E2 -8791.82} C_VEL
LIN {X 0,Y 446.428,Z 202.18,A -85,B 0,C 180,E1 -8794.846,E2 -8794.846} C_VEL
LIN {X 0,Y 446.454,Z 202.182,A -85,B 0,C 180,E1 -8798.232,E2 -8798.232} C_VEL
LIN {X 0,Y 446.425,Z 202.181,A -85,B 0,C 180,E1 -8801.648,E2 -8801.648} C_VEL
LIN {X 0,Y 446.475,Z 202.183,A -85,B 0,C 180,E1 -8804.479,E2 -8804.479} C_VEL
LIN {X 0,Y 446.509,Z 202.153,A -85,B 0,C 180,E1 -8808.193,E2 -8808.193} C_VEL
LIN {X 0,Y 446.567,Z 202.168,A -85,B 0,C 180,E1 -8811.858,E2 -8811.858} C_VEL
LIN {X 0,Y 446.618,Z 202.153,A -85,B 0,C 180,E1 -8814.583,E2 -8814.583} C_VEL
LIN {X 0,Y 446.676,Z 202.141,A -85,B 0,C 180,E1 -8817.295,E2 -8817.295} C_VEL
LIN {X 0,Y 446.759,Z 202.143,A -85,B 0,C 180,E1 -8820,E2 -8820} C_VEL
LIN {X 0,Y 446.676,Z 202.153,A -85,B 0,C 180,E1 -8822.706,E2 -8822.706} C_VEL
LIN {X 0,Y 446.615,Z 202.158,A -85,B 0,C 180,E1 -8826.325,E2 -8826.325} C_VEL
LIN {X 0,Y 446.507,Z 202.174,A -85,B 0,C 180,E1 -8829.056,E2 -8829.056} C_VEL
LIN {X 0,Y 446.49,Z 202.171,A -85,B 0,C 180,E1 -8832.731,E2 -8832.731} C_VEL
LIN {X 0,Y 446.489,Z 202.18,A -85,B 0,C 180,E1 -8836.24,E2 -8836.24} C_VEL
LIN {X 0,Y 446.44,Z 202.172,A -85,B 0,C 180,E1 -8839.305,E2 -8839.305} C_VEL
LIN {X 0,Y 446.393,Z 202.192,A -85,B 0,C 180,E1 -8842.201,E2 -8842.201} C_VEL
LIN {X 0,Y 446.43,Z 202.174,A -85,B 0,C 180,E1 -8845.155,E2 -8845.155} C_VEL
LIN {X 0,Y 446.459,Z 202.181,A -85,B 0,C 180,E1 -8848.181,E2 -8848.181} C_VEL
LIN {X 0,Y 446.394,Z 202.186,A -85,B 0,C 180,E1 -8851.777,E2 -8851.777} C_VEL
LIN {X 0,Y 446.407,Z 202.189,A -85,B 0,C 180,E1 -8854.526,E2 -8854.526} C_VEL
LIN {X 0,Y 446.391,Z 202.189,A -85,B 0,C 180,E1 -8858.082,E2 -8858.082} C_VEL
LIN {X 0,Y 446.408,Z 202.187,A -85,B 0,C 180,E1 -8861.394,E2 -8861.394} C_VEL
LIN {X 0,Y 446.432,Z 202.174,A -85,B 0,C 180,E1 -8865.107,E2 -8865.107} C_VEL
LIN {X 0,Y 446.403,Z 202.189,A -85,B 0,C 180,E1 -8868.611,E2 -8868.611} C_VEL
LIN {X 0,Y 446.412,Z 202.19,A -85,B 0,C 180,E1 -8872.126,E2 -8872.126} C_VEL
LIN {X 0,Y 446.418,Z 202.181,A -85,B 0,C 180,E1 -8875.48,E2 -8875.48} C_VEL
LIN {X 0,Y 446.405,Z 202.188,A -85,B 0,C 180,E1 -8878.703,E2 -8878.703} C_VEL
LIN {X 0,Y 446.442,Z 202.187,A -85,B 0,C 180,E1 -8881.833,E2 -8881.833} C_VEL
LIN {X 0,Y 446.431,Z 202.184,A -85,B 0,C 180,E1 -8884.85,E2 -8884.85} C_VEL
LIN {X 0,Y 446.444,Z 202.186,A -85,B 0,C 180,E1 -8888.248,E2 -8888.248} C_VEL
LIN {X 0,Y 446.438,Z 202.186,A -85,B 0,C 180,E1 -8891.651,E2 -8891.651} C_VEL
LIN {X 0,Y 446.459,Z 202.186,A -85,B 0,C 180,E1 -8894.481,E2 -8894.481} C_VEL
LIN {X 0,Y 446.517,Z 202.178,A -85,B 0,C 180,E1 -8897.387,E2 -8897.387} C_VEL
LIN {X 0,Y 446.527,Z 202.176,A -85,B 0,C 180,E1 -8900.947,E2 -8900.947} C_VEL
LIN {X 0,Y 446.609,Z 202.161,A -85,B 0,C 180,E1 -8903.678,E2 -8903.678} C_VEL
LIN {X 0,Y 446.556,Z 202.277,A -85,B 0,C 180,E1 -8905.065,E2 -8905.065} C_VEL
LIN {X 0,Y 447.581,Z 206.038,A -85,B 0,C 180,E1 -8905.648,E2 -8905.648} C_VEL
LIN {X 0,Y 448.357,Z 208.835,A -85,B 0,C 180,E1 -8905.974,E2 -8905.974} C_VEL
LIN {X 0,Y 449.169,Z 212.157,A -85,B 0,C 180,E1 -8906.209,E2 -8906.209} C_VEL
LIN {X 0,Y 450.614,Z 219.583,A -85,B 0,C 180,E1 -8906.506,E2 -8906.506} C_VEL
LIN {X 0,Y 452.595,Z 231.38,A -85,B 0,C 180,E1 -8906.868,E2 -8906.868} C_VEL
LIN {X 0,Y 453.829,Z 235.058,A -85,B 0,C 180,E1 -8907.024,E2 -8907.024} C_VEL
LIN {X 0,Y 455.215,Z 238.267,A -85,B 0,C 180,E1 -8907.181,E2 -8907.181} C_VEL
LIN {X 0,Y 451.872,Z 415.953,A -85,B 0,C 180,E1 -8910.169,E2 -8910.169} C_VEL
LIN {X 0,Y 451.155,Z 433,A -85,B 0,C 180,E1 -8910.644,E2 -8910.644} C_VEL
LIN {X 0,Y 450.305,Z 448.829,A -85,B 0,C 180,E1 -8911.268,E2 -8911.268} C_VEL
LIN {X 0,Y 449.268,Z 463.704,A -85,B 0,C 180,E1 -8912.019,E2 -8912.019} C_VEL
LIN {X 0,Y 448.125,Z 478.21,A -85,B 0,C 180,E1 -8912.924,E2 -8912.924} C_VEL
LIN {X 0,Y 446.731,Z 493.124,A -85,B 0,C 180,E1 -8914.062,E2 -8914.062} C_VEL
LIN {X 0,Y 445.38,Z 506.802,A -85,B 0,C 180,E1 -8915.321,E2 -8915.321} C_VEL
LIN {X 0,Y 444.211,Z 518.513,A -85,B 0,C 180,E1 -8916.589,E2 -8916.589} C_VEL
LIN {X 0,Y 443.011,Z 529.635,A -85,B 0,C 180,E1 -8917.981,E2 -8917.981} C_VEL
LIN {X 0,Y 441.785,Z 541.229,A -85,B 0,C 180,E1 -8919.698,E2 -8919.698} C_VEL
LIN {X 0,Y 440.753,Z 551.478,A -85,B 0,C 180,E1 -8921.499,E2 -8921.499} C_VEL
LIN {X 0,Y 439.956,Z 560.335,A -85,B 0,C 180,E1 -8923.348,E2 -8923.348} C_VEL
LIN {X 0,Y 439.328,Z 568.157,A -85,B 0,C 180,E1 -8925.306,E2 -8925.306} C_VEL
LIN {X 0,Y 438.853,Z 574.438,A -85,B 0,C 180,E1 -8927.235,E2 -8927.235} C_VEL
LIN {X 0,Y 438.614,Z 579.112,A -85,B 0,C 180,E1 -8929.025,E2 -8929.025} C_VEL
LIN {X 0,Y 438.377,Z 582.526,A -85,B 0,C 180,E1 -8930.654,E2 -8930.654} C_VEL
LIN {X 0,Y 438.163,Z 585.586,A -85,B 0,C 180,E1 -8932.642,E2 -8932.642} C_VEL
LIN {X 0,Y 438.078,Z 587.569,A -85,B 0,C 180,E1 -8934.654,E2 -8934.654} C_VEL
LIN {X 0,Y 438.093,Z 588.335,A -85,B 0,C 180,E1 -8936.693,E2 -8936.693} C_VEL
LIN {X 0,Y 438.119,Z 587.949,A -85,B 0,C 180,E1 -8938.768,E2 -8938.768} C_VEL
LIN {X 0,Y 438.224,Z 586.35,A -85,B 0,C 180,E1 -8940.878,E2 -8940.878} C_VEL
LIN {X 0,Y 438.358,Z 583.377,A -85,B 0,C 180,E1 -8943.033,E2 -8943.033} C_VEL
LIN {X 0,Y 438.588,Z 578.892,A -85,B 0,C 180,E1 -8945.232,E2 -8945.232} C_VEL
LIN {X 0,Y 438.94,Z 573.894,A -85,B 0,C 180,E1 -8947.1,E2 -8947.1} C_VEL
LIN {X 0,Y 439.477,Z 566.982,A -85,B 0,C 180,E1 -8949.175,E2 -8949.175} C_VEL
LIN {X 0,Y 440.129,Z 558.949,A -85,B 0,C 180,E1 -8951.14,E2 -8951.14} C_VEL
LIN {X 0,Y 441.151,Z 548.471,A -85,B 0,C 180,E1 -8953.239,E2 -8953.239} C_VEL
LIN {X 0,Y 442.286,Z 537.861,A -85,B 0,C 180,E1 -8955.001,E2 -8955.001} C_VEL
LIN {X 0,Y 443.41,Z 527.392,A -85,B 0,C 180,E1 -8956.483,E2 -8956.483} C_VEL
LIN {X 0,Y 444.717,Z 515.185,A -85,B 0,C 180,E1 -8957.967,E2 -8957.967} C_VEL
LIN {X 0,Y 446.029,Z 502.459,A -85,B 0,C 180,E1 -8959.284,E2 -8959.284} C_VEL
LIN {X 0,Y 447.396,Z 488.433,A -85,B 0,C 180,E1 -8960.495,E2 -8960.495} C_VEL
LIN {X 0,Y 448.727,Z 473.755,A -85,B 0,C 180,E1 -8961.546,E2 -8961.546} C_VEL
LIN {X 0,Y 449.983,Z 457.811,A -85,B 0,C 180,E1 -8962.474,E2 -8962.474} C_VEL
LIN {X 0,Y 450.992,Z 441.687,A -85,B 0,C 180,E1 -8963.211,E2 -8963.211} C_VEL
LIN {X 0,Y 451.876,Z 425.071,A -85,B 0,C 180,E1 -8963.771,E2 -8963.771} C_VEL
LIN {X 0,Y 452.428,Z 407.526,A -85,B 0,C 180,E1 -8964.163,E2 -8964.163} C_VEL
LIN {X 0,Y 455.681,Z 239.098,A -85,B 0,C 180,E1 -8967,E2 -8967} C_VEL
LIN {X 0,Y 454.733,Z 236.456,A -85,B 0,C 180,E1 -8967.121,E2 -8967.121} C_VEL
LIN {X 0,Y 446.477,Z 219.531,A -85,B 0,C 180,E1 -8968.091,E2 -8968.091} C_VEL
LIN {X 0,Y 441.671,Z 210.213,A -85,B 0,C 180,E1 -8968.692,E2 -8968.692} C_VEL
LIN {X 0,Y 439.39,Z 203.063,A -85,B 0,C 180,E1 -8969.937,E2 -8969.937} C_VEL
LIN {X 0,Y 439.443,Z 203.061,A -85,B 0,C 180,E1 -8972.367,E2 -8972.367} C_VEL
LIN {X 0,Y 439.413,Z 203.063,A -85,B 0,C 180,E1 -8975.736,E2 -8975.736} C_VEL
LIN {X 0,Y 439.39,Z 203.059,A -85,B 0,C 180,E1 -8979.397,E2 -8979.397} C_VEL
LIN {X 0,Y 439.433,Z 203.052,A -85,B 0,C 180,E1 -8982.309,E2 -8982.309} C_VEL
LIN {X 0,Y 439.448,Z 203.056,A -85,B 0,C 180,E1 -8985.173,E2 -8985.173} C_VEL
LIN {X 0,Y 439.484,Z 203.056,A -85,B 0,C 180,E1 -8988.001,E2 -8988.001} C_VEL
LIN {X 0,Y 439.548,Z 203.045,A -85,B 0,C 180,E1 -8991.726,E2 -8991.726} C_VEL
LIN {X 0,Y 439.619,Z 203.035,A -85,B 0,C 180,E1 -8994.495,E2 -8994.495} C_VEL
LIN {X 0,Y 439.632,Z 203.033,A -85,B 0,C 180,E1 -8998.167,E2 -8998.167} C_VEL
LIN {X 0,Y 439.76,Z 203.021,A -85,B 0,C 180,E1 -9000,E2 -9000} C_VEL
LIN {X 0,Y 439.638,Z 203.032,A -85,B 0,C 180,E1 -9002.748,E2 -9002.748} C_VEL
LIN {X 0,Y 439.603,Z 203.036,A -85,B 0,C 180,E1 -9006.425,E2 -9006.425} C_VEL
LIN {X 0,Y 439.495,Z 203.053,A -85,B 0,C 180,E1 -9009.201,E2 -9009.201} C_VEL
LIN {X 0,Y 439.465,Z 203.054,A -85,B 0,C 180,E1 -9012.937,E2 -9012.937} C_VEL
LIN {X 0,Y 439.446,Z 203.053,A -85,B 0,C 180,E1 -9016.347,E2 -9016.347} C_VEL
LIN {X 0,Y 439.401,Z 203.065,A -85,B 0,C 180,E1 -9019.626,E2 -9019.626} C_VEL
LIN {X 0,Y 439.363,Z 203.065,A -85,B 0,C 180,E1 -9022.575,E2 -9022.575} C_VEL
LIN {X 0,Y 439.397,Z 203.065,A -85,B 0,C 180,E1 -9025.585,E2 -9025.585} C_VEL
LIN {X 0,Y 439.417,Z 203.061,A -85,B 0,C 180,E1 -9028.673,E2 -9028.673} C_VEL
LIN {X 0,Y 439.365,Z 203.064,A -85,B 0,C 180,E1 -9032.029,E2 -9032.029} C_VEL
LIN {X 0,Y 439.392,Z 203.067,A -85,B 0,C 180,E1 -9035.339,E2 -9035.339} C_VEL
LIN {X 0,Y 439.376,Z 203.066,A -85,B 0,C 180,E1 -9038.595,E2 -9038.595} C_VEL
LIN {X 0,Y 439.381,Z 203.059,A -85,B 0,C 180,E1 -9041.255,E2 -9041.255} C_VEL
LIN {X 0,Y 439.377,Z 203.063,A -85,B 0,C 180,E1 -9044.732,E2 -9044.732} C_VEL
LIN {X 0,Y 439.359,Z 203.065,A -85,B 0,C 180,E1 -9047.79,E2 -9047.79} C_VEL
LIN {X 0,Y 439.359,Z 203.066,A -85,B 0,C 180,E1 -9050.219,E2 -9050.219} C_VEL
LIN {X 0,Y 439.373,Z 203.069,A -85,B 0,C 180,E1 -9053.712,E2 -9053.712} C_VEL
LIN {X 0,Y 439.405,Z 203.173,A -85,B 0,C 180,E1 -9054.726,E2 -9054.726} C_VEL
LIN {X 0,Y 444.621,Z 218.966,A -85,B 0,C 180,E1 -9057.175,E2 -9057.175} C_VEL
LIN {X 0,Y 448.288,Z 231.081,A -85,B 0,C 180,E1 -9058.914,E2 -9058.914} C_VEL
LIN {X 0,Y 451.298,Z 238.106,A -85,B 0,C 180,E1 -9059.284,E2 -9059.284} C_VEL
LIN {X 0,Y 455.379,Z 262.284,A -85,B 0,C 180,E1 -9060.043,E2 -9060.043} C_VEL
LIN {X 0,Y 451.936,Z 438.471,A -85,B 0,C 180,E1 -9063.024,E2 -9063.024} C_VEL
LIN {X 0,Y 451.152,Z 454.556,A -85,B 0,C 180,E1 -9063.454,E2 -9063.454} C_VEL
LIN {X 0,Y 450.215,Z 469.719,A -85,B 0,C 180,E1 -9064.018,E2 -9064.018} C_VEL
LIN {X 0,Y 449.071,Z 485.077,A -85,B 0,C 180,E1 -9064.755,E2 -9064.755} C_VEL
LIN {X 0,Y 447.824,Z 500.144,A -85,B 0,C 180,E1 -9065.672,E2 -9065.672} C_VEL
LIN {X 0,Y 446.472,Z 514.089,A -85,B 0,C 180,E1 -9066.702,E2 -9066.702} C_VEL
LIN {X 0,Y 445.029,Z 528.448,A -85,B 0,C 180,E1 -9067.97,E2 -9067.97} C_VEL
LIN {X 0,Y 443.809,Z 540.625,A -85,B 0,C 180,E1 -9069.238,E2 -9069.238} C_VEL
LIN {X 0,Y 442.492,Z 552.977,A -85,B 0,C 180,E1 -9070.756,E2 -9070.756} C_VEL
LIN {X 0,Y 441.318,Z 564.264,A -85,B 0,C 180,E1 -9072.386,E2 -9072.386} C_VEL
LIN {X 0,Y 440.402,Z 575.209,A -85,B 0,C 180,E1 -9074.257,E2 -9074.257} C_VEL
LIN {X 0,Y 439.582,Z 584.414,A -85,B 0,C 180,E1 -9076.122,E2 -9076.122} C_VEL
LIN {X 0,Y 439.089,Z 592.125,A -85,B 0,C 180,E1 -9077.989,E2 -9077.989} C_VEL
LIN {X 0,Y 438.563,Z 599.869,A -85,B 0,C 180,E1 -9080.311,E2 -9080.311} C_VEL
LIN {X 0,Y 438.389,Z 605.768,A -85,B 0,C 180,E1 -9082.63,E2 -9082.63} C_VEL
LIN {X 0,Y 438.308,Z 609.222,A -85,B 0,C 180,E1 -9084.477,E2 -9084.477} C_VEL
LIN {X 0,Y 438.23,Z 611.734,A -85,B 0,C 180,E1 -9086.32,E2 -9086.32} C_VEL
LIN {X 0,Y 438.289,Z 613.157,A -85,B 0,C 180,E1 -9088.16,E2 -9088.16} C_VEL
LIN {X 0,Y 438.248,Z 613.696,A -85,B 0,C 180,E1 -9089.998,E2 -9089.998} C_VEL
LIN {X 0,Y 438.289,Z 613.172,A -85,B 0,C 180,E1 -9091.836,E2 -9091.836} C_VEL
LIN {X 0,Y 438.229,Z 611.762,A -85,B 0,C 180,E1 -9093.676,E2 -9093.676} C_VEL
LIN {X 0,Y 438.305,Z 609.267,A -85,B 0,C 180,E1 -9095.518,E2 -9095.518} C_VEL
LIN {X 0,Y 438.385,Z 605.825,A -85,B 0,C 180,E1 -9097.366,E2 -9097.366} C_VEL
LIN {X 0,Y 438.566,Z 599.938,A -85,B 0,C 180,E1 -9099.684,E2 -9099.684} C_VEL
LIN {X 0,Y 438.936,Z 593.865,A -85,B 0,C 180,E1 -9101.543,E2 -9101.543} C_VEL
LIN {X 0,Y 439.409,Z 586.526,A -85,B 0,C 180,E1 -9103.407,E2 -9103.407} C_VEL
LIN {X 0,Y 440.111,Z 577.755,A -85,B 0,C 180,E1 -9105.274,E2 -9105.274} C_VEL
LIN {X 0,Y 440.994,Z 567.986,A -85,B 0,C 180,E1 -9107.021,E2 -9107.021} C_VEL
LIN {X 0,Y 441.925,Z 558.018,A -85,B 0,C 180,E1 -9108.543,E2 -9108.543} C_VEL
LIN {X 0,Y 443.237,Z 545.547,A -85,B 0,C 180,E1 -9110.171,E2 -9110.171} C_VEL
LIN {X 0,Y 444.5,Z 533.008,A -85,B 0,C 180,E1 -9111.565,E2 -9111.565} C_VEL
LIN {X 0,Y 445.866,Z 519.389,A -85,B 0,C 180,E1 -9112.836,E2 -9112.836} C_VEL
LIN {X 0,Y 447.163,Z 506.199,A -85,B 0,C 180,E1 -9113.87,E2 -9113.87} C_VEL
LIN {X 0,Y 448.46,Z 491.52,A -85,B 0,C 180,E1 -9114.834,E2 -9114.834} C_VEL
LIN {X 0,Y 449.633,Z 476.406,A -85,B 0,C 180,E1 -9115.64,E2 -9115.64} C_VEL
LIN {X 0,Y 450.597,Z 460.516,A -85,B 0,C 180,E1 -9116.295,E2 -9116.295} C_VEL
LIN {X 0,Y 451.435,Z 444.629,A -85,B 0,C 180,E1 -9116.772,E2 -9116.772} C_VEL
LIN {X 0,Y 452.068,Z 425.025,A -85,B 0,C 180,E1 -9117.156,E2 -9117.156} C_VEL
LIN {X 0,Y 454.957,Z 261.504,A -85,B 0,C 180,E1 -9119.889,E2 -9119.889} C_VEL
LIN {X 0,Y 450.56,Z 236.797,A -85,B 0,C 180,E1 -9120.654,E2 -9120.654} C_VEL
LIN {X 0,Y 448.228,Z 231.554,A -85,B 0,C 180,E1 -9120.93,E2 -9120.93} C_VEL
LIN {X 0,Y 443.299,Z 215.233,A -85,B 0,C 180,E1 -9123.251,E2 -9123.251} C_VEL
LIN {X 0,Y 439.375,Z 203.066,A -85,B 0,C 180,E1 -9125.108,E2 -9125.108} C_VEL
LIN {X 0,Y 439.358,Z 203.071,A -85,B 0,C 180,E1 -9128.593,E2 -9128.593} C_VEL
LIN {X 0,Y 439.367,Z 203.072,A -85,B 0,C 180,E1 -9131.254,E2 -9131.254} C_VEL
LIN {X 0,Y 439.38,Z 203.068,A -85,B 0,C 180,E1 -9134.727,E2 -9134.727} C_VEL
LIN {X 0,Y 439.375,Z 203.066,A -85,B 0,C 180,E1 -9137.794,E2 -9137.794} C_VEL
LIN {X 0,Y 439.425,Z 203.056,A -85,B 0,C 180,E1 -9140.228,E2 -9140.228} C_VEL
LIN {X 0,Y 439.35,Z 203.062,A -85,B 0,C 180,E1 -9143.711,E2 -9143.711} C_VEL
LIN {X 0,Y 439.344,Z 203.064,A -85,B 0,C 180,E1 -9147.052,E2 -9147.052} C_VEL
LIN {X 0,Y 439.353,Z 203.068,A -85,B 0,C 180,E1 -9150.272,E2 -9150.272} C_VEL
LIN {X 0,Y 439.398,Z 203.049,A -85,B 0,C 180,E1 -9153.395,E2 -9153.395} C_VEL
LIN {X 0,Y 439.363,Z 203.067,A -85,B 0,C 180,E1 -9156.429,E2 -9156.429} C_VEL
LIN {X 0,Y 439.382,Z 203.05,A -85,B 0,C 180,E1 -9159.397,E2 -9159.397} C_VEL
LIN {X 0,Y 439.399,Z 203.057,A -85,B 0,C 180,E1 -9162.309,E2 -9162.309} C_VEL
LIN {X 0,Y 439.416,Z 203.056,A -85,B 0,C 180,E1 -9165.173,E2 -9165.173} C_VEL
LIN {X 0,Y 439.477,Z 203.027,A -85,B 0,C 180,E1 -9168.002,E2 -9168.002} C_VEL
LIN {X 0,Y 439.515,Z 203.046,A -85,B 0,C 180,E1 -9171.726,E2 -9171.726} C_VEL
LIN {X 0,Y 439.593,Z 203.029,A -85,B 0,C 180,E1 -9174.496,E2 -9174.496} C_VEL
LIN {X 0,Y 439.604,Z 203.023,A -85,B 0,C 180,E1 -9178.168,E2 -9178.168} C_VEL
LIN {X 0,Y 439.73,Z 203.018,A -85,B 0,C 180,E1 -9180,E2 -9180} C_VEL
LIN {X 0,Y 439.623,Z 203.03,A -85,B 0,C 180,E1 -9182.749,E2 -9182.749} C_VEL
LIN {X 0,Y 439.586,Z 203.034,A -85,B 0,C 180,E1 -9186.426,E2 -9186.426} C_VEL
LIN {X 0,Y 439.469,Z 203.05,A -85,B 0,C 180,E1 -9189.203,E2 -9189.203} C_VEL
LIN {X 0,Y 439.434,Z 203.053,A -85,B 0,C 180,E1 -9192.939,E2 -9192.939} C_VEL
LIN {X 0,Y 439.43,Z 203.061,A -85,B 0,C 180,E1 -9196.356,E2 -9196.356} C_VEL
LIN {X 0,Y 439.374,Z 203.052,A -85,B 0,C 180,E1 -9199.628,E2 -9199.628} C_VEL
LIN {X 0,Y 439.339,Z 203.073,A -85,B 0,C 180,E1 -9202.577,E2 -9202.577} C_VEL
LIN {X 0,Y 439.378,Z 203.052,A -85,B 0,C 180,E1 -9205.587,E2 -9205.587} C_VEL
LIN {X 0,Y 439.391,Z 203.066,A -85,B 0,C 180,E1 -9208.676,E2 -9208.676} C_VEL
LIN {X 0,Y 439.345,Z 203.063,A -85,B 0,C 180,E1 -9212.033,E2 -9212.033} C_VEL
LIN {X 0,Y 439.373,Z 203.063,A -85,B 0,C 180,E1 -9215.343,E2 -9215.343} C_VEL
LIN {X 0,Y 439.349,Z 203.058,A -85,B 0,C 180,E1 -9218.599,E2 -9218.599} C_VEL
LIN {X 0,Y 439.368,Z 203.063,A -85,B 0,C 180,E1 -9221.26,E2 -9221.26} C_VEL
LIN {X 0,Y 439.38,Z 203.054,A -85,B 0,C 180,E1 -9224.733,E2 -9224.733} C_VEL
LIN {X 0,Y 439.368,Z 203.067,A -85,B 0,C 180,E1 -9227.797,E2 -9227.797} C_VEL
LIN {X 0,Y 439.374,Z 203.06,A -85,B 0,C 180,E1 -9230.226,E2 -9230.226} C_VEL
LIN {X 0,Y 439.364,Z 203.068,A -85,B 0,C 180,E1 -9233.716,E2 -9233.716} C_VEL
LIN {X 0,Y 439.362,Z 203.065,A -85,B 0,C 180,E1 -9237.057,E2 -9237.057} C_VEL
LIN {X 0,Y 439.368,Z 203.063,A -85,B 0,C 180,E1 -9240.277,E2 -9240.277} C_VEL
LIN {X 0,Y 439.373,Z 203.065,A -85,B 0,C 180,E1 -9243.396,E2 -9243.396} C_VEL
LIN {X 0,Y 439.376,Z 203.065,A -85,B 0,C 180,E1 -9246.432,E2 -9246.432} C_VEL
LIN {X 0,Y 439.382,Z 203.066,A -85,B 0,C 180,E1 -9249.4,E2 -9249.4} C_VEL
LIN {X 0,Y 439.387,Z 203.067,A -85,B 0,C 180,E1 -9252.311,E2 -9252.311} C_VEL
LIN {X 0,Y 439.401,Z 203.064,A -85,B 0,C 180,E1 -9255.175,E2 -9255.175} C_VEL
LIN {X 0,Y 439.483,Z 203.053,A -85,B 0,C 180,E1 -9258.004,E2 -9258.004} C_VEL
LIN {X 0,Y 439.503,Z 203.052,A -85,B 0,C 180,E1 -9261.728,E2 -9261.728} C_VEL
LIN {X 0,Y 439.592,Z 203.197,A -85,B 0,C 180,E1 -9264.613,E2 -9264.613} C_VEL
LIN {X 0,Y 441.459,Z 209.789,A -85,B 0,C 180,E1 -9265.631,E2 -9265.631} C_VEL
LIN {X 0,Y 448.85,Z 224.333,A -85,B 0,C 180,E1 -9266.464,E2 -9266.464} C_VEL
LIN {X 0,Y 453.829,Z 235.058,A -85,B 0,C 180,E1 -9267.024,E2 -9267.024} C_VEL
LIN {X 0,Y 454.292,Z 238.103,A -85,B 0,C 180,E1 -9267.113,E2 -9267.113} C_VEL
LIN {X 0,Y 453.297,Z 242.586,A -85,B 0,C 180,E1 -9267.124,E2 -9267.124} C_VEL
LIN {X 0,Y 449.439,Z 251.599,A -85,B 0,C 180,E1 -9267.012,E2 -9267.012} C_VEL
LIN {X 0,Y 448.68,Z 255.726,A -85,B 0,C 180,E1 -9267.033,E2 -9267.033} C_VEL
LIN {X 0,Y 445.505,Z 415.261,A -85,B 0,C 180,E1 -9269.748,E2 -9269.748} C_VEL
LIN {X 0,Y 444.846,Z 431.635,A -85,B 0,C 180,E1 -9270.2,E2 -9270.2} C_VEL
LIN {X 0,Y 444.004,Z 447.096,A -85,B 0,C 180,E1 -9270.796,E2 -9270.796} C_VEL
LIN {X 0,Y 442.926,Z 462.008,A -85,B 0,C 180,E1 -9271.531,E2 -9271.531} C_VEL
LIN {X 0,Y 441.642,Z 477.721,A -85,B 0,C 180,E1 -9272.51,E2 -9272.51} C_VEL
LIN {X 0,Y 440.191,Z 492.733,A -85,B 0,C 180,E1 -9273.664,E2 -9273.664} C_VEL
LIN {X 0,Y 438.758,Z 506.525,A -85,B 0,C 180,E1 -9274.941,E2 -9274.941} C_VEL
LIN {X 0,Y 437.499,Z 518.363,A -85,B 0,C 180,E1 -9276.231,E2 -9276.231} C_VEL
LIN {X 0,Y 436.265,Z 529.477,A -85,B 0,C 180,E1 -9277.639,E2 -9277.639} C_VEL
LIN {X 0,Y 435.02,Z 540.619,A -85,B 0,C 180,E1 -9279.299,E2 -9279.299} C_VEL
LIN {X 0,Y 433.987,Z 550.201,A -85,B 0,C 180,E1 -9280.971,E2 -9280.971} C_VEL
LIN {X 0,Y 433.195,Z 558.411,A -85,B 0,C 180,E1 -9282.643,E2 -9282.643} C_VEL
LIN {X 0,Y 432.459,Z 566.404,A -85,B 0,C 180,E1 -9284.591,E2 -9284.591} C_VEL
LIN {X 0,Y 431.921,Z 573.19,A -85,B 0,C 180,E1 -9286.601,E2 -9286.601} C_VEL
LIN {X 0,Y 431.592,Z 578.447,A -85,B 0,C 180,E1 -9288.516,E2 -9288.516} C_VEL
LIN {X 0,Y 431.397,Z 581.686,A -85,B 0,C 180,E1 -9290.007,E2 -9290.007} C_VEL
LIN {X 0,Y 431.129,Z 585.102,A -85,B 0,C 180,E1 -9292.022,E2 -9292.022} C_VEL
LIN {X 0,Y 431.014,Z 587.311,A -85,B 0,C 180,E1 -9294.058,E2 -9294.058} C_VEL
LIN {X 0,Y 431.002,Z 588.463,A -85,B 0,C 180,E1 -9296.253,E2 -9296.253} C_VEL
LIN {X 0,Y 431.022,Z 588.4,A -85,B 0,C 180,E1 -9298.297,E2 -9298.297} C_VEL
LIN {X 0,Y 431.103,Z 587.103,A -85,B 0,C 180,E1 -9300.357,E2 -9300.357} C_VEL
LIN {X 0,Y 431.213,Z 584.5,A -85,B 0,C 180,E1 -9302.538,E2 -9302.538} C_VEL
LIN {X 0,Y 431.454,Z 580.469,A -85,B 0,C 180,E1 -9304.76,E2 -9304.76} C_VEL
LIN {X 0,Y 431.734,Z 576.385,A -85,B 0,C 180,E1 -9306.454,E2 -9306.454} C_VEL
LIN {X 0,Y 432.288,Z 569.551,A -85,B 0,C 180,E1 -9308.705,E2 -9308.705} C_VEL
LIN {X 0,Y 432.941,Z 561.606,A -85,B 0,C 180,E1 -9310.798,E2 -9310.798} C_VEL
LIN {X 0,Y 433.741,Z 553.541,A -85,B 0,C 180,E1 -9312.57,E2 -9312.57} C_VEL
LIN {X 0,Y 434.867,Z 543.722,A -85,B 0,C 180,E1 -9314.38,E2 -9314.38} C_VEL
LIN {X 0,Y 436.078,Z 532.478,A -85,B 0,C 180,E1 -9316.131,E2 -9316.131} C_VEL
LIN {X 0,Y 437.43,Z 520.931,A -85,B 0,C 180,E1 -9317.652,E2 -9317.652} C_VEL
LIN {X 0,Y 438.89,Z 508.017,A -85,B 0,C 180,E1 -9319.101,E2 -9319.101} C_VEL
LIN {X 0,Y 440.254,Z 495.26,A -85,B 0,C 180,E1 -9320.316,E2 -9320.316} C_VEL
LIN {X 0,Y 441.618,Z 481.535,A -85,B 0,C 180,E1 -9321.408,E2 -9321.408} C_VEL
LIN {X 0,Y 442.961,Z 466.135,A -85,B 0,C 180,E1 -9322.423,E2 -9322.423} C_VEL
LIN {X 0,Y 444.126,Z 450.876,A -85,B 0,C 180,E1 -9323.23,E2 -9323.23} C_VEL
LIN {X 0,Y 445.109,Z 434.899,A -85,B 0,C 180,E1 -9323.885,E2 -9323.885} C_VEL
LIN {X 0,Y 445.785,Z 418.697,A -85,B 0,C 180,E1 -9324.36,E2 -9324.36} C_VEL
LIN {X 0,Y 446.374,Z 393.266,A -85,B 0,C 180,E1 -9324.835,E2 -9324.835} C_VEL
LIN {X 0,Y 449.538,Z 240.559,A -85,B 0,C 180,E1 -9327.446,E2 -9327.446} C_VEL
LIN {X 0,Y 440.353,Z 221.697,A -85,B 0,C 180,E1 -9328.554,E2 -9328.554} C_VEL
LIN {X 0,Y 434.474,Z 210.454,A -85,B 0,C 180,E1 -9329.312,E2 -9329.312} C_VEL
LIN {X 0,Y 432.334,Z 203.946,A -85,B 0,C 180,E1 -9330.477,E2 -9330.477} C_VEL
LIN {X 0,Y 432.402,Z 203.934,A -85,B 0,C 180,E1 -9333.373,E2 -9333.373} C_VEL
LIN {X 0,Y 432.37,Z 203.938,A -85,B 0,C 180,E1 -9336.023,E2 -9336.023} C_VEL
LIN {X 0,Y 432.352,Z 203.936,A -85,B 0,C 180,E1 -9339.046,E2 -9339.046} C_VEL
LIN {X 0,Y 432.379,Z 203.932,A -85,B 0,C 180,E1 -9342.011,E2 -9342.011} C_VEL
LIN {X 0,Y 432.396,Z 203.934,A -85,B 0,C 180,E1 -9344.926,E2 -9344.926} C_VEL
LIN {X 0,Y 432.46,Z 203.929,A -85,B 0,C 180,E1 -9347.803,E2 -9347.803} C_VEL
LIN {X 0,Y 432.492,Z 203.924,A -85,B 0,C 180,E1 -9351.59,E2 -9351.59} C_VEL
LIN {X 0,Y 432.595,Z 203.911,A -85,B 0,C 180,E1 -9354.406,E2 -9354.406} C_VEL
LIN {X 0,Y 432.602,Z 203.909,A -85,B 0,C 180,E1 -9358.138,E2 -9358.138} C_VEL
LIN {X 0,Y 432.73,Z 203.897,A -85,B 0,C 180,E1 -9360,E2 -9360} C_VEL
LIN {X 0,Y 432.59,Z 203.91,A -85,B 0,C 180,E1 -9362.793,E2 -9362.793} C_VEL
LIN {X 0,Y 432.553,Z 203.914,A -85,B 0,C 180,E1 -9366.53,E2 -9366.53} C_VEL
LIN {X 0,Y 432.439,Z 203.933,A -85,B 0,C 180,E1 -9369.353,E2 -9369.353} C_VEL
LIN {X 0,Y 432.431,Z 203.929,A -85,B 0,C 180,E1 -9372.803,E2 -9372.803} C_VEL
LIN {X 0,Y 432.411,Z 203.93,A -85,B 0,C 180,E1 -9376.478,E2 -9376.478} C_VEL
LIN {X 0,Y 432.337,Z 203.943,A -85,B 0,C 180,E1 -9379.96,E2 -9379.96} C_VEL
LIN {X 0,Y 432.317,Z 203.946,A -85,B 0,C 180,E1 -9382.964,E2 -9382.964} C_VEL
LIN {X 0,Y 432.36,Z 203.938,A -85,B 0,C 180,E1 -9386.032,E2 -9386.032} C_VEL
LIN {X 0,Y 432.342,Z 203.943,A -85,B 0,C 180,E1 -9389.187,E2 -9389.187} C_VEL
LIN {X 0,Y 432.321,Z 203.942,A -85,B 0,C 180,E1 -9392.443,E2 -9392.443} C_VEL
LIN {X 0,Y 432.337,Z 203.942,A -85,B 0,C 180,E1 -9395.817,E2 -9395.817} C_VEL
LIN {X 0,Y 432.327,Z 203.947,A -85,B 0,C 180,E1 -9399.345,E2 -9399.345} C_VEL
LIN {X 0,Y 432.325,Z 203.94,A -85,B 0,C 180,E1 -9401.798,E2 -9401.798} C_VEL
LIN {X 0,Y 432.333,Z 203.94,A -85,B 0,C 180,E1 -9404.347,E2 -9404.347} C_VEL
LIN {X 0,Y 432.308,Z 203.947,A -85,B 0,C 180,E1 -9407.017,E2 -9407.017} C_VEL
LIN {X 0,Y 432.309,Z 203.947,A -85,B 0,C 180,E1 -9409.824,E2 -9409.824} C_VEL
LIN {X 0,Y 432.305,Z 203.947,A -85,B 0,C 180,E1 -9413.021,E2 -9413.021} C_VEL
LIN {X 0,Y 432.363,Z 204.109,A -85,B 0,C 180,E1 -9414.184,E2 -9414.184} C_VEL
LIN {X 0,Y 437.517,Z 219.505,A -85,B 0,C 180,E1 -9416.646,E2 -9416.646} C_VEL
LIN {X 0,Y 440.999,Z 230.736,A -85,B 0,C 180,E1 -9418.316,E2 -9418.316} C_VEL
LIN {X 0,Y 445.432,Z 240.492,A -85,B 0,C 180,E1 -9418.866,E2 -9418.866} C_VEL
LIN {X 0,Y 449.211,Z 262.964,A -85,B 0,C 180,E1 -9419.591,E2 -9419.591} C_VEL
LIN {X 0,Y 445.653,Z 437.792,A -85,B 0,C 180,E1 -9422.593,E2 -9422.593} C_VEL
LIN {X 0,Y 444.838,Z 453.678,A -85,B 0,C 180,E1 -9423.016,E2 -9423.016} C_VEL
LIN {X 0,Y 443.842,Z 469.67,A -85,B 0,C 180,E1 -9423.617,E2 -9423.617} C_VEL
LIN {X 0,Y 442.639,Z 484.967,A -85,B 0,C 180,E1 -9424.362,E2 -9424.362} C_VEL
LIN {X 0,Y 441.237,Z 501.025,A -85,B 0,C 180,E1 -9425.358,E2 -9425.358} C_VEL
LIN {X 0,Y 439.739,Z 515.348,A -85,B 0,C 180,E1 -9426.448,E2 -9426.448} C_VEL
LIN {X 0,Y 438.236,Z 529.448,A -85,B 0,C 180,E1 -9427.735,E2 -9427.735} C_VEL
LIN {X 0,Y 436.85,Z 542.341,A -85,B 0,C 180,E1 -9429.13,E2 -9429.13} C_VEL
LIN {X 0,Y 435.487,Z 554.547,A -85,B 0,C 180,E1 -9430.679,E2 -9430.679} C_VEL
LIN {X 0,Y 434.299,Z 565.64,A -85,B 0,C 180,E1 -9432.346,E2 -9432.346} C_VEL
LIN {X 0,Y 433.474,Z 575.016,A -85,B 0,C 180,E1 -9433.999,E2 -9433.999} C_VEL
LIN {X 0,Y 432.566,Z 584.213,A -85,B 0,C 180,E1 -9435.893,E2 -9435.893} C_VEL
LIN {X 0,Y 432.047,Z 591.921,A -85,B 0,C 180,E1 -9437.79,E2 -9437.79} C_VEL
LIN {X 0,Y 431.486,Z 599.666,A -85,B 0,C 180,E1 -9440.151,E2 -9440.151} C_VEL
LIN {X 0,Y 431.309,Z 605.566,A -85,B 0,C 180,E1 -9442.508,E2 -9442.508} C_VEL
LIN {X 0,Y 431.221,Z 609.019,A -85,B 0,C 180,E1 -9444.386,E2 -9444.386} C_VEL
LIN {X 0,Y 431.138,Z 611.53,A -85,B 0,C 180,E1 -9446.259,E2 -9446.259} C_VEL
LIN {X 0,Y 431.212,Z 612.954,A -85,B 0,C 180,E1 -9448.13,E2 -9448.13} C_VEL
LIN {X 0,Y 431.162,Z 613.492,A -85,B 0,C 180,E1 -9449.998,E2 -9449.998} C_VEL
LIN {X 0,Y 431.211,Z 612.966,A -85,B 0,C 180,E1 -9451.866,E2 -9451.866} C_VEL
LIN {X 0,Y 431.137,Z 611.553,A -85,B 0,C 180,E1 -9453.736,E2 -9453.736} C_VEL
LIN {X 0,Y 431.218,Z 609.055,A -85,B 0,C 180,E1 -9455.609,E2 -9455.609} C_VEL
LIN {X 0,Y 431.305,Z 605.607,A -85,B 0,C 180,E1 -9457.488,E2 -9457.488} C_VEL
LIN {X 0,Y 431.487,Z 599.712,A -85,B 0,C 180,E1 -9459.845,E2 -9459.845} C_VEL
LIN {X 0,Y 431.907,Z 593.633,A -85,B 0,C 180,E1 -9461.733,E2 -9461.733} C_VEL
LIN {X 0,Y 432.403,Z 586.283,A -85,B 0,C 180,E1 -9463.628,E2 -9463.628} C_VEL
LIN {X 0,Y 433.163,Z 577.502,A -85,B 0,C 180,E1 -9465.525,E2 -9465.525} C_VEL
LIN {X 0,Y 434.162,Z 567.089,A -85,B 0,C 180,E1 -9467.41,E2 -9467.41} C_VEL
LIN {X 0,Y 435.298,Z 556.094,A -85,B 0,C 180,E1 -9469.08,E2 -9469.08} C_VEL
LIN {X 0,Y 436.673,Z 543.269,A -85,B 0,C 180,E1 -9470.734,E2 -9470.734} C_VEL
LIN {X 0,Y 438.036,Z 530.302,A -85,B 0,C 180,E1 -9472.147,E2 -9472.147} C_VEL
LIN {X 0,Y 439.559,Z 516.274,A -85,B 0,C 180,E1 -9473.432,E2 -9473.432} C_VEL
LIN {X 0,Y 441.066,Z 500.897,A -85,B 0,C 180,E1 -9474.601,E2 -9474.601} C_VEL
LIN {X 0,Y 442.464,Z 484.951,A -85,B 0,C 180,E1 -9475.581,E2 -9475.581} C_VEL
LIN {X 0,Y 443.63,Z 469.446,A -85,B 0,C 180,E1 -9476.329,E2 -9476.329} C_VEL
LIN {X 0,Y 444.562,Z 453.065,A -85,B 0,C 180,E1 -9476.934,E2 -9476.934} C_VEL
LIN {X 0,Y 445.393,Z 436.169,A -85,B 0,C 180,E1 -9477.36,E2 -9477.36} C_VEL
LIN {X 0,Y 448.77,Z 263.192,A -85,B 0,C 180,E1 -9480.297,E2 -9480.297} C_VEL
LIN {X 0,Y 444.679,Z 239.515,A -85,B 0,C 180,E1 -9481.038,E2 -9481.038} C_VEL
LIN {X 0,Y 440.929,Z 231.279,A -85,B 0,C 180,E1 -9481.491,E2 -9481.491} C_VEL
LIN {X 0,Y 435.308,Z 213.031,A -85,B 0,C 180,E1 -9484.166,E2 -9484.166} C_VEL
LIN {X 0,Y 432.323,Z 203.943,A -85,B 0,C 180,E1 -9485.581,E2 -9485.581} C_VEL
LIN {X 0,Y 432.32,Z 203.948,A -85,B 0,C 180,E1 -9488.712,E2 -9488.712} C_VEL
LIN {X 0,Y 432.312,Z 203.945,A -85,B 0,C 180,E1 -9491.795,E2 -9491.795} C_VEL
LIN {X 0,Y 432.312,Z 203.946,A -85,B 0,C 180,E1 -9494.345,E2 -9494.345} C_VEL
LIN {X 0,Y 432.302,Z 203.949,A -85,B 0,C 180,E1 -9497.013,E2 -9497.013} C_VEL
LIN {X 0,Y 432.331,Z 203.941,A -85,B 0,C 180,E1 -9499.815,E2 -9499.815} C_VEL
LIN {X 0,Y 432.29,Z 203.942,A -85,B 0,C 180,E1 -9503.021,E2 -9503.021} C_VEL
LIN {X 0,Y 432.332,Z 203.942,A -85,B 0,C 180,E1 -9505.995,E2 -9505.995} C_VEL
LIN {X 0,Y 432.319,Z 203.946,A -85,B 0,C 180,E1 -9509.488,E2 -9509.488} C_VEL
LIN {X 0,Y 432.361,Z 203.93,A -85,B 0,C 180,E1 -9512.927,E2 -9512.927} C_VEL
LIN {X 0,Y 432.344,Z 203.94,A -85,B 0,C 180,E1 -9516.022,E2 -9516.022} C_VEL
LIN {X 0,Y 432.346,Z 203.93,A -85,B 0,C 180,E1 -9519.046,E2 -9519.046} C_VEL
LIN {X 0,Y 432.346,Z 203.934,A -85,B 0,C 180,E1 -9522.01,E2 -9522.01} C_VEL
LIN {X 0,Y 432.364,Z 203.938,A -85,B 0,C 180,E1 -9524.926,E2 -9524.926} C_VEL
LIN {X 0,Y 432.449,Z 203.901,A -85,B 0,C 180,E1 -9527.804,E2 -9527.804} C_VEL
LIN {X 0,Y 432.46,Z 203.926,A -85,B 0,C 180,E1 -9531.59,E2 -9531.59} C_VEL
LIN {X 0,Y 432.569,Z 203.905,A -85,B 0,C 180,E1 -9534.406,E2 -9534.406} C_VEL
LIN {X 0,Y 432.574,Z 203.898,A -85,B 0,C 180,E1 -9538.138,E2 -9538.138} C_VEL
LIN {X 0,Y 432.7,Z 203.894,A -85,B 0,C 180,E1 -9540,E2 -9540} C_VEL
LIN {X 0,Y 432.573,Z 203.908,A -85,B 0,C 180,E1 -9542.794,E2 -9542.794} C_VEL
LIN {X 0,Y 432.541,Z 203.913,A -85,B 0,C 180,E1 -9546.531,E2 -9546.531} C_VEL
LIN {X 0,Y 432.412,Z 203.928,A -85,B 0,C 180,E1 -9549.354,E2 -9549.354} C_VEL
LIN {X 0,Y 432.4,Z 203.926,A -85,B 0,C 180,E1 -9552.805,E2 -9552.805} C_VEL
LIN {X 0,Y 432.393,Z 203.935,A -85,B 0,C 180,E1 -9556.485,E2 -9556.485} C_VEL
LIN {X 0,Y 432.31,Z 203.933,A -85,B 0,C 180,E1 -9559.962,E2 -9559.962} C_VEL
LIN {X 0,Y 432.293,Z 203.946,A -85,B 0,C 180,E1 -9562.966,E2 -9562.966} C_VEL
LIN {X 0,Y 432.337,Z 203.929,A -85,B 0,C 180,E1 -9566.035,E2 -9566.035} C_VEL
LIN {X 0,Y 432.317,Z 203.943,A -85,B 0,C 180,E1 -9569.19,E2 -9569.19} C_VEL
LIN {X 0,Y 432.299,Z 203.936,A -85,B 0,C 180,E1 -9572.446,E2 -9572.446} C_VEL
LIN {X 0,Y 432.322,Z 203.942,A -85,B 0,C 180,E1 -9575.635,E2 -9575.635} C_VEL
LIN {X 0,Y 432.312,Z 203.933,A -85,B 0,C 180,E1 -9578.716,E2 -9578.716} C_VEL
LIN {X 0,Y 432.313,Z 203.945,A -85,B 0,C 180,E1 -9581.8,E2 -9581.8} C_VEL
LIN {X 0,Y 432.316,Z 203.937,A -85,B 0,C 180,E1 -9584.35,E2 -9584.35} C_VEL
LIN {X 0,Y 432.3,Z 203.945,A -85,B 0,C 180,E1 -9587.019,E2 -9587.019} C_VEL
LIN {X 0,Y 432.299,Z 203.944,A -85,B 0,C 180,E1 -9589.827,E2 -9589.827} C_VEL
LIN {X 0,Y 432.302,Z 203.946,A -85,B 0,C 180,E1 -9593.026,E2 -9593.026} C_VEL
LIN {X 0,Y 432.349,Z 203.935,A -85,B 0,C 180,E1 -9596,E2 -9596} C_VEL
LIN {X 0,Y 432.337,Z 203.94,A -85,B 0,C 180,E1 -9599.493,E2 -9599.493} C_VEL
LIN {X 0,Y 432.339,Z 203.944,A -85,B 0,C 180,E1 -9601.877,E2 -9601.877} C_VEL
LIN {X 0,Y 432.371,Z 203.938,A -85,B 0,C 180,E1 -9605.542,E2 -9605.542} C_VEL
LIN {X 0,Y 432.345,Z 203.942,A -85,B 0,C 180,E1 -9609.049,E2 -9609.049} C_VEL
LIN {X 0,Y 432.347,Z 203.947,A -85,B 0,C 180,E1 -9612.013,E2 -9612.013} C_VEL
LIN {X 0,Y 432.349,Z 203.942,A -85,B 0,C 180,E1 -9614.928,E2 -9614.928} C_VEL
LIN {X 0,Y 432.459,Z 203.929,A -85,B 0,C 180,E1 -9617.806,E2 -9617.806} C_VEL
LIN {X 0,Y 432.464,Z 203.93,A -85,B 0,C 180,E1 -9621.592,E2 -9621.592} C_VEL
LIN {X 0,Y 432.558,Z 203.961,A -85,B 0,C 180,E1 -9624.116,E2 -9624.116} C_VEL
LIN {X 0,Y 434.272,Z 210.057,A -85,B 0,C 180,E1 -9625.07,E2 -9625.07} C_VEL
LIN {X 0,Y 443.496,Z 228.253,A -85,B 0,C 180,E1 -9626.137,E2 -9626.137} C_VEL
LIN {X 0,Y 449.009,Z 240.56,A -85,B 0,C 180,E1 -9626.776,E2 -9626.776} C_VEL
LIN {X 0,Y 448.68,Z 255.726,A -85,B 0,C 180,E1 -9627.033,E2 -9627.033} C_VEL
LIN {X 0,Y 447.99,Z 261.582,A -85,B 0,C 180,E1 -9627.091,E2 -9627.091} C_VEL
LIN {X 0,Y 442.503,Z 280.67,A -85,B 0,C 180,E1 -9627.048,E2 -9627.048} C_VEL
LIN {X 0,Y 441.854,Z 286.522,A -85,B 0,C 180,E1 -9627.111,E2 -9627.111} C_VEL
LIN {X 0,Y 439.179,Z 415.764,A -85,B 0,C 180,E1 -9629.343,E2 -9629.343} C_VEL
LIN {X 0,Y 438.436,Z 432.947,A -85,B 0,C 180,E1 -9629.83,E2 -9629.83} C_VEL
LIN {X 0,Y 437.506,Z 448.74,A -85,B 0,C 180,E1 -9630.462,E2 -9630.462} C_VEL
LIN {X 0,Y 436.323,Z 463.975,A -85,B 0,C 180,E1 -9631.246,E2 -9631.246} C_VEL
LIN {X 0,Y 435.052,Z 478.852,A -85,B 0,C 180,E1 -9632.201,E2 -9632.201} C_VEL
LIN {X 0,Y 433.531,Z 493.754,A -85,B 0,C 180,E1 -9633.371,E2 -9633.371} C_VEL
LIN {X 0,Y 432.029,Z 507.415,A -85,B 0,C 180,E1 -9634.667,E2 -9634.667} C_VEL
LIN {X 0,Y 430.666,Z 519.683,A -85,B 0,C 180,E1 -9636.044,E2 -9636.044} C_VEL
LIN {X 0,Y 429.334,Z 531.055,A -85,B 0,C 180,E1 -9637.527,E2 -9637.527} C_VEL
LIN {X 0,Y 428.05,Z 542.013,A -85,B 0,C 180,E1 -9639.214,E2 -9639.214} C_VEL
LIN {X 0,Y 426.968,Z 551.403,A -85,B 0,C 180,E1 -9640.913,E2 -9640.913} C_VEL
LIN {X 0,Y 426.051,Z 560.219,A -85,B 0,C 180,E1 -9642.789,E2 -9642.789} C_VEL
LIN {X 0,Y 425.326,Z 568.251,A -85,B 0,C 180,E1 -9644.842,E2 -9644.842} C_VEL
LIN {X 0,Y 424.8,Z 574.416,A -85,B 0,C 180,E1 -9646.782,E2 -9646.782} C_VEL
LIN {X 0,Y 424.48,Z 579.603,A -85,B 0,C 180,E1 -9648.812,E2 -9648.812} C_VEL
LIN {X 0,Y 424.237,Z 582.753,A -85,B 0,C 180,E1 -9650.36,E2 -9650.36} C_VEL
LIN {X 0,Y 423.989,Z 585.879,A -85,B 0,C 180,E1 -9652.412,E2 -9652.412} C_VEL
LIN {X 0,Y 423.891,Z 587.913,A -85,B 0,C 180,E1 -9654.489,E2 -9654.489} C_VEL
LIN {X 0,Y 423.901,Z 588.728,A -85,B 0,C 180,E1 -9656.594,E2 -9656.594} C_VEL
LIN {X 0,Y 423.948,Z 588.41,A -85,B 0,C 180,E1 -9658.736,E2 -9658.736} C_VEL
LIN {X 0,Y 424.046,Z 586.879,A -85,B 0,C 180,E1 -9660.918,E2 -9660.918} C_VEL
LIN {X 0,Y 424.182,Z 583.942,A -85,B 0,C 180,E1 -9663.146,E2 -9663.146} C_VEL
LIN {X 0,Y 424.503,Z 579.534,A -85,B 0,C 180,E1 -9665.413,E2 -9665.413} C_VEL
LIN {X 0,Y 424.867,Z 574.342,A -85,B 0,C 180,E1 -9667.438,E2 -9667.438} C_VEL
LIN {X 0,Y 425.477,Z 567.653,A -85,B 0,C 180,E1 -9669.524,E2 -9669.524} C_VEL
LIN {X 0,Y 426.105,Z 560.787,A -85,B 0,C 180,E1 -9671.281,E2 -9671.281} C_VEL
LIN {X 0,Y 426.989,Z 552.474,A -85,B 0,C 180,E1 -9673.085,E2 -9673.085} C_VEL
LIN {X 0,Y 428.223,Z 542.655,A -85,B 0,C 180,E1 -9674.888,E2 -9674.888} C_VEL
LIN {X 0,Y 429.535,Z 531.164,A -85,B 0,C 180,E1 -9676.673,E2 -9676.673} C_VEL
LIN {X 0,Y 430.951,Z 519.457,A -85,B 0,C 180,E1 -9678.202,E2 -9678.202} C_VEL
LIN {X 0,Y 432.513,Z 506.293,A -85,B 0,C 180,E1 -9679.662,E2 -9679.662} C_VEL
LIN {X 0,Y 434.105,Z 491.934,A -85,B 0,C 180,E1 -9680.997,E2 -9680.997} C_VEL
LIN {X 0,Y 435.515,Z 478.107,A -85,B 0,C 180,E1 -9682.071,E2 -9682.071} C_VEL
LIN {X 0,Y 436.903,Z 462.476,A -85,B 0,C 180,E1 -9683.061,E2 -9683.061} C_VEL
LIN {X 0,Y 438.077,Z 446.825,A -85,B 0,C 180,E1 -9683.841,E2 -9683.841} C_VEL
LIN {X 0,Y 439.022,Z 430.622,A -85,B 0,C 180,E1 -9684.457,E2 -9684.457} C_VEL
LIN {X 0,Y 439.719,Z 414.237,A -85,B 0,C 180,E1 -9684.895,E2 -9684.895} C_VEL
LIN {X 0,Y 443.516,Z 243.428,A -85,B 0,C 180,E1 -9687.87,E2 -9687.87} C_VEL
LIN {X 0,Y 442.584,Z 240.834,A -85,B 0,C 180,E1 -9687.995,E2 -9687.995} C_VEL
LIN {X 0,Y 434.259,Z 223.998,A -85,B 0,C 180,E1 -9689.03,E2 -9689.03} C_VEL
LIN {X 0,Y 427.243,Z 210.779,A -85,B 0,C 180,E1 -9689.954,E2 -9689.954} C_VEL
LIN {X 0,Y 425.317,Z 204.817,A -85,B 0,C 180,E1 -9691.045,E2 -9691.045} C_VEL
LIN {X 0,Y 425.357,Z 204.811,A -85,B 0,C 180,E1 -9693.505,E2 -9693.505} C_VEL
LIN {X 0,Y 425.287,Z 204.82,A -85,B 0,C 180,E1 -9696.633,E2 -9696.633} C_VEL
LIN {X 0,Y 425.297,Z 204.815,A -85,B 0,C 180,E1 -9699.694,E2 -9699.694} C_VEL
LIN {X 0,Y 425.344,Z 204.806,A -85,B 0,C 180,E1 -9702.697,E2 -9702.697} C_VEL
LIN {X 0,Y 425.349,Z 204.814,A -85,B 0,C 180,E1 -9705.65,E2 -9705.65} C_VEL
LIN {X 0,Y 425.35,Z 204.813,A -85,B 0,C 180,E1 -9708.563,E2 -9708.563} C_VEL
LIN {X 0,Y 425.54,Z 204.791,A -85,B 0,C 180,E1 -9712.407,E2 -9712.407} C_VEL
LIN {X 0,Y 425.552,Z 204.789,A -85,B 0,C 180,E1 -9714.313,E2 -9714.313} C_VEL
LIN {X 0,Y 425.571,Z 204.785,A -85,B 0,C 180,E1 -9718.107,E2 -9718.107} C_VEL
LIN {X 0,Y 425.7,Z 204.773,A -85,B 0,C 180,E1 -9720,E2 -9720} C_VEL
LIN {X 0,Y 425.543,Z 204.788,A -85,B 0,C 180,E1 -9722.839,E2 -9722.839} C_VEL
LIN {X 0,Y 425.545,Z 204.792,A -85,B 0,C 180,E1 -9725.686,E2 -9725.686} C_VEL
LIN {X 0,Y 425.408,Z 204.805,A -85,B 0,C 180,E1 -9728.55,E2 -9728.55} C_VEL
LIN {X 0,Y 425.412,Z 204.803,A -85,B 0,C 180,E1 -9732.401,E2 -9732.401} C_VEL
LIN {X 0,Y 425.387,Z 204.805,A -85,B 0,C 180,E1 -9736.311,E2 -9736.311} C_VEL
LIN {X 0,Y 425.328,Z 204.818,A -85,B 0,C 180,E1 -9739.635,E2 -9739.635} C_VEL
LIN {X 0,Y 425.304,Z 204.821,A -85,B 0,C 180,E1 -9743.365,E2 -9743.365} C_VEL
LIN {X 0,Y 425.346,Z 204.813,A -85,B 0,C 180,E1 -9746.843,E2 -9746.843} C_VEL
LIN {X 0,Y 425.29,Z 204.82,A -85,B 0,C 180,E1 -9749.719,E2 -9749.719} C_VEL
LIN {X 0,Y 425.269,Z 204.826,A -85,B 0,C 180,E1 -9753.049,E2 -9753.049} C_VEL
LIN {X 0,Y 425.281,Z 204.82,A -85,B 0,C 180,E1 -9755.928,E2 -9755.928} C_VEL
LIN {X 0,Y 425.282,Z 204.824,A -85,B 0,C 180,E1 -9759.04,E2 -9759.04} C_VEL
LIN {X 0,Y 425.283,Z 204.818,A -85,B 0,C 180,E1 -9761.956,E2 -9761.956} C_VEL
LIN {X 0,Y 425.284,Z 204.82,A -85,B 0,C 180,E1 -9765.283,E2 -9765.283} C_VEL
LIN {X 0,Y 425.254,Z 204.827,A -85,B 0,C 180,E1 -9768.618,E2 -9768.618} C_VEL
LIN {X 0,Y 425.285,Z 204.823,A -85,B 0,C 180,E1 -9771.099,E2 -9771.099} C_VEL
LIN {X 0,Y 425.316,Z 204.948,A -85,B 0,C 180,E1 -9773.599,E2 -9773.599} C_VEL
LIN {X 0,Y 430.885,Z 221.495,A -85,B 0,C 180,E1 -9776.318,E2 -9776.318} C_VEL
LIN {X 0,Y 433.711,Z 230.477,A -85,B 0,C 180,E1 -9777.69,E2 -9777.69} C_VEL
LIN {X 0,Y 439.697,Z 243.311,A -85,B 0,C 180,E1 -9778.454,E2 -9778.454} C_VEL
LIN {X 0,Y 443.148,Z 264.581,A -85,B 0,C 180,E1 -9779.146,E2 -9779.146} C_VEL
LIN {X 0,Y 439.366,Z 438.233,A -85,B 0,C 180,E1 -9782.172,E2 -9782.172} C_VEL
LIN {X 0,Y 438.473,Z 454.617,A -85,B 0,C 180,E1 -9782.624,E2 -9782.624} C_VEL
LIN {X 0,Y 437.375,Z 470.923,A -85,B 0,C 180,E1 -9783.26,E2 -9783.26} C_VEL
LIN {X 0,Y 436.034,Z 486.867,A -85,B 0,C 180,E1 -9784.073,E2 -9784.073} C_VEL
LIN {X 0,Y 434.648,Z 501.84,A -85,B 0,C 180,E1 -9785.031,E2 -9785.031} C_VEL
LIN {X 0,Y 433.038,Z 516.656,A -85,B 0,C 180,E1 -9786.188,E2 -9786.188} C_VEL
LIN {X 0,Y 431.468,Z 530.471,A -85,B 0,C 180,E1 -9787.492,E2 -9787.492} C_VEL
LIN {X 0,Y 430.002,Z 543.283,A -85,B 0,C 180,E1 -9788.925,E2 -9788.925} C_VEL
LIN {X 0,Y 428.7,Z 554.358,A -85,B 0,C 180,E1 -9790.361,E2 -9790.361} C_VEL
LIN {X 0,Y 427.423,Z 565.537,A -85,B 0,C 180,E1 -9792.066,E2 -9792.066} C_VEL
LIN {X 0,Y 426.517,Z 574.823,A -85,B 0,C 180,E1 -9793.731,E2 -9793.731} C_VEL
LIN {X 0,Y 425.562,Z 584.019,A -85,B 0,C 180,E1 -9795.656,E2 -9795.656} C_VEL
LIN {X 0,Y 425.023,Z 591.728,A -85,B 0,C 180,E1 -9797.585,E2 -9797.585} C_VEL
LIN {X 0,Y 424.429,Z 599.468,A -85,B 0,C 180,E1 -9799.985,E2 -9799.985} C_VEL
LIN {X 0,Y 424.226,Z 605.364,A -85,B 0,C 180,E1 -9802.382,E2 -9802.382} C_VEL
LIN {X 0,Y 424.141,Z 608.817,A -85,B 0,C 180,E1 -9804.292,E2 -9804.292} C_VEL
LIN {X 0,Y 424.051,Z 611.327,A -85,B 0,C 180,E1 -9806.197,E2 -9806.197} C_VEL
LIN {X 0,Y 424.136,Z 612.751,A -85,B 0,C 180,E1 -9808.099,E2 -9808.099} C_VEL
LIN {X 0,Y 424.079,Z 613.287,A -85,B 0,C 180,E1 -9809.998,E2 -9809.998} C_VEL
LIN {X 0,Y 424.136,Z 612.759,A -85,B 0,C 180,E1 -9811.897,E2 -9811.897} C_VEL
LIN {X 0,Y 424.049,Z 611.342,A -85,B 0,C 180,E1 -9813.799,E2 -9813.799} C_VEL
LIN {X 0,Y 424.221,Z 607.948,A -85,B 0,C 180,E1 -9816.278,E2 -9816.278} C_VEL
LIN {X 0,Y 424.272,Z 603.225,A -85,B 0,C 180,E1 -9818.571,E2 -9818.571} C_VEL
LIN {X 0,Y 424.53,Z 598.042,A -85,B 0,C 180,E1 -9820.49,E2 -9820.49} C_VEL
LIN {X 0,Y 425.002,Z 591.716,A -85,B 0,C 180,E1 -9822.411,E2 -9822.411} C_VEL
LIN {X 0,Y 425.652,Z 582.957,A -85,B 0,C 180,E1 -9824.581,E2 -9824.581} C_VEL
LIN {X 0,Y 426.621,Z 573.499,A -85,B 0,C 180,E1 -9826.506,E2 -9826.506} C_VEL
LIN {X 0,Y 427.558,Z 563.731,A -85,B 0,C 180,E1 -9828.196,E2 -9828.196} C_VEL
LIN {X 0,Y 428.877,Z 552.346,A -85,B 0,C 180,E1 -9829.875,E2 -9829.875} C_VEL
LIN {X 0,Y 430.254,Z 540.253,A -85,B 0,C 180,E1 -9831.399,E2 -9831.399} C_VEL
LIN {X 0,Y 431.682,Z 527.599,A -85,B 0,C 180,E1 -9832.744,E2 -9832.744} C_VEL
LIN {X 0,Y 433.241,Z 513.029,A -85,B 0,C 180,E1 -9834.049,E2 -9834.049} C_VEL
LIN {X 0,Y 434.675,Z 498.644,A -85,B 0,C 180,E1 -9835.12,E2 -9835.12} C_VEL
LIN {X 0,Y 436.166,Z 483.406,A -85,B 0,C 180,E1 -9836.042,E2 -9836.042} C_VEL
LIN {X 0,Y 437.332,Z 467.642,A -85,B 0,C 180,E1 -9836.802,E2 -9836.802} C_VEL
LIN {X 0,Y 438.305,Z 451.534,A -85,B 0,C 180,E1 -9837.383,E2 -9837.383} C_VEL
LIN {X 0,Y 439.114,Z 434.708,A -85,B 0,C 180,E1 -9837.797,E2 -9837.797} C_VEL
LIN {X 0,Y 442.561,Z 263.793,A -85,B 0,C 180,E1 -9840.74,E2 -9840.74} C_VEL
LIN {X 0,Y 438.734,Z 242.108,A -85,B 0,C 180,E1 -9841.439,E2 -9841.439} C_VEL
LIN {X 0,Y 433.603,Z 231.005,A -85,B 0,C 180,E1 -9842.072,E2 -9842.072} C_VEL
LIN {X 0,Y 428.291,Z 213.972,A -85,B 0,C 180,E1 -9844.635,E2 -9844.635} C_VEL
LIN {X 0,Y 425.27,Z 204.825,A -85,B 0,C 180,E1 -9846.092,E2 -9846.092} C_VEL
LIN {X 0,Y 425.263,Z 204.827,A -85,B 0,C 180,E1 -9849.038,E2 -9849.038} C_VEL
LIN {X 0,Y 425.269,Z 204.821,A -85,B 0,C 180,E1 -9851.956,E2 -9851.956} C_VEL
LIN {X 0,Y 425.267,Z 204.819,A -85,B 0,C 180,E1 -9855.28,E2 -9855.28} C_VEL
LIN {X 0,Y 425.281,Z 204.819,A -85,B 0,C 180,E1 -9858.623,E2 -9858.623} C_VEL
LIN {X 0,Y 425.297,Z 204.824,A -85,B 0,C 180,E1 -9861.102,E2 -9861.102} C_VEL
LIN {X 0,Y 425.274,Z 204.818,A -85,B 0,C 180,E1 -9864.662,E2 -9864.662} C_VEL
LIN {X 0,Y 425.236,Z 204.812,A -85,B 0,C 180,E1 -9868.071,E2 -9868.071} C_VEL
LIN {X 0,Y 425.302,Z 204.819,A -85,B 0,C 180,E1 -9871.366,E2 -9871.366} C_VEL
LIN {X 0,Y 425.265,Z 204.811,A -85,B 0,C 180,E1 -9874.553,E2 -9874.553} C_VEL
LIN {X 0,Y 425.292,Z 204.818,A -85,B 0,C 180,E1 -9877.718,E2 -9877.718} C_VEL
LIN {X 0,Y 425.334,Z 204.798,A -85,B 0,C 180,E1 -9880.703,E2 -9880.703} C_VEL
LIN {X 0,Y 425.356,Z 204.811,A -85,B 0,C 180,E1 -9883.687,E2 -9883.687} C_VEL
LIN {X 0,Y 425.398,Z 204.779,A -85,B 0,C 180,E1 -9887.598,E2 -9887.598} C_VEL
LIN {X 0,Y 425.411,Z 204.805,A -85,B 0,C 180,E1 -9891.45,E2 -9891.45} C_VEL
LIN {X 0,Y 425.544,Z 204.781,A -85,B 0,C 180,E1 -9894.314,E2 -9894.314} C_VEL
LIN {X 0,Y 425.544,Z 204.773,A -85,B 0,C 180,E1 -9898.108,E2 -9898.108} C_VEL
LIN {X 0,Y 425.67,Z 204.77,A -85,B 0,C 180,E1 -9900,E2 -9900} C_VEL
LIN {X 0,Y 425.524,Z 204.785,A -85,B 0,C 180,E1 -9902.841,E2 -9902.841} C_VEL
LIN {X 0,Y 425.498,Z 204.792,A -85,B 0,C 180,E1 -9906.64,E2 -9906.64} C_VEL
LIN {X 0,Y 425.37,Z 204.805,A -85,B 0,C 180,E1 -9909.511,E2 -9909.511} C_VEL
LIN {X 0,Y 425.362,Z 204.804,A -85,B 0,C 180,E1 -9912.905,E2 -9912.905} C_VEL
LIN {X 0,Y 425.34,Z 204.811,A -85,B 0,C 180,E1 -9916.61,E2 -9916.61} C_VEL
LIN {X 0,Y 425.3,Z 204.804,A -85,B 0,C 180,E1 -9919.638,E2 -9919.638} C_VEL
LIN {X 0,Y 425.28,Z 204.818,A -85,B 0,C 180,E1 -9923.367,E2 -9923.367} C_VEL
LIN {X 0,Y 425.321,Z 204.808,A -85,B 0,C 180,E1 -9926.846,E2 -9926.846} C_VEL
LIN {X 0,Y 425.265,Z 204.823,A -85,B 0,C 180,E1 -9929.722,E2 -9929.722} C_VEL
LIN {X 0,Y 425.258,Z 204.812,A -85,B 0,C 180,E1 -9933.051,E2 -9933.051} C_VEL
LIN {X 0,Y 425.26,Z 204.824,A -85,B 0,C 180,E1 -9935.932,E2 -9935.932} C_VEL
LIN {X 0,Y 425.255,Z 204.809,A -85,B 0,C 180,E1 -9939.043,E2 -9939.043} C_VEL
LIN {X 0,Y 425.27,Z 204.824,A -85,B 0,C 180,E1 -9941.961,E2 -9941.961} C_VEL
LIN {X 0,Y 425.267,Z 204.809,A -85,B 0,C 180,E1 -9945.286,E2 -9945.286} C_VEL
LIN {X 0,Y 425.249,Z 204.824,A -85,B 0,C 180,E1 -9948.623,E2 -9948.623} C_VEL
LIN {X 0,Y 425.277,Z 204.814,A -85,B 0,C 180,E1 -9951.104,E2 -9951.104} C_VEL
LIN {X 0,Y 425.288,Z 204.813,A -85,B 0,C 180,E1 -9954.667,E2 -9954.667} C_VEL
LIN {X 0,Y 425.256,Z 204.829,A -85,B 0,C 180,E1 -9958.076,E2 -9958.076} C_VEL
LIN {X 0,Y 425.305,Z 204.816,A -85,B 0,C 180,E1 -9961.37,E2 -9961.37} C_VEL
LIN {X 0,Y 425.263,Z 204.821,A -85,B 0,C 180,E1 -9964.556,E2 -9964.556} C_VEL
LIN {X 0,Y 425.278,Z 204.819,A -85,B 0,C 180,E1 -9966.637,E2 -9966.637} C_VEL
LIN {X 0,Y 425.291,Z 204.825,A -85,B 0,C 180,E1 -9969.698,E2 -9969.698} C_VEL
LIN {X 0,Y 425.294,Z 204.82,A -85,B 0,C 180,E1 -9972.699,E2 -9972.699} C_VEL
LIN {X 0,Y 425.327,Z 204.817,A -85,B 0,C 180,E1 -9975.652,E2 -9975.652} C_VEL
LIN {X 0,Y 425.349,Z 204.813,A -85,B 0,C 180,E1 -9978.567,E2 -9978.567} C_VEL
LIN {X 0,Y 425.408,Z 204.81,A -85,B 0,C 180,E1 -9981.452,E2 -9981.452} C_VEL
LIN {X 0,Y 425.501,Z 204.931,A -85,B 0,C 180,E1 -9983.631,E2 -9983.631} C_VEL
LIN {X 0,Y 427.123,Z 210.12,A -85,B 0,C 180,E1 -9984.488,E2 -9984.488} C_VEL
LIN {X 0,Y 438.255,Z 232.399,A -85,B 0,C 180,E1 -9985.815,E2 -9985.815} C_VEL
LIN {X 0,Y 442.743,Z 242.154,A -85,B 0,C 180,E1 -9986.342,E2 -9986.342} C_VEL
LIN {X 0,Y 441.854,Z 286.522,A -85,B 0,C 180,E1 -9987.111,E2 -9987.111} C_VEL
LIN {X 0,Y 441.2,Z 292.374,A -85,B 0,C 180,E1 -9987.173,E2 -9987.173} C_VEL
LIN {X 0,Y 435.677,Z 311.452,A -85,B 0,C 180,E1 -9987.13,E2 -9987.13} C_VEL
LIN {X 0,Y 434.989,Z 317.307,A -85,B 0,C 180,E1 -9987.19,E2 -9987.19} C_VEL
LIN {X 0,Y 432.863,Z 416.094,A -85,B 0,C 180,E1 -9988.927,E2 -9988.927} C_VEL
LIN {X 0,Y 432.079,Z 433.248,A -85,B 0,C 180,E1 -9989.42,E2 -9989.42} C_VEL
LIN {X 0,Y 431.094,Z 449.048,A -85,B 0,C 180,E1 -9990.061,E2 -9990.061} C_VEL
LIN {X 0,Y 429.917,Z 463.72,A -85,B 0,C 180,E1 -9990.822,E2 -9990.822} C_VEL
LIN {X 0,Y 428.58,Z 478.93,A -85,B 0,C 180,E1 -9991.808,E2 -9991.808} C_VEL
LIN {X 0,Y 427.044,Z 493.339,A -85,B 0,C 180,E1 -9992.95,E2 -9992.95} C_VEL
LIN {X 0,Y 425.477,Z 507.117,A -85,B 0,C 180,E1 -9994.265,E2 -9994.265} C_VEL
LIN {X 0,Y 423.86,Z 520.668,A -85,B 0,C 180,E1 -9995.808,E2 -9995.808} C_VEL
LIN {X 0,Y 422.401,Z 532.555,A -85,B 0,C 180,E1 -9997.411,E2 -9997.411} C_VEL
LIN {X 0,Y 421.086,Z 543.384,A -85,B 0,C 180,E1 -9999.125,E2 -9999.125} C_VEL
LIN {X 0,Y 419.814,Z 553.854,A -85,B 0,C 180,E1 -10001.102,E2 -10001.102} C_VEL
LIN {X 0,Y 418.95,Z 561.982,A -85,B 0,C 180,E1 -10002.941,E2 -10002.941} C_VEL
LIN {X 0,Y 418.18,Z 569.947,A -85,B 0,C 180,E1 -10005.101,E2 -10005.101} C_VEL
LIN {X 0,Y 417.65,Z 576.035,A -85,B 0,C 180,E1 -10007.128,E2 -10007.128} C_VEL
LIN {X 0,Y 417.297,Z 581.397,A -85,B 0,C 180,E1 -10009.413,E2 -10009.413} C_VEL
LIN {X 0,Y 416.987,Z 585.354,A -85,B 0,C 180,E1 -10011.766,E2 -10011.766} C_VEL
LIN {X 0,Y 416.841,Z 587.633,A -85,B 0,C 180,E1 -10013.87,E2 -10013.87} C_VEL
LIN {X 0,Y 416.792,Z 588.832,A -85,B 0,C 180,E1 -10016.004,E2 -10016.004} C_VEL
LIN {X 0,Y 416.827,Z 588.845,A -85,B 0,C 180,E1 -10018.172,E2 -10018.172} C_VEL
LIN {X 0,Y 416.92,Z 587.602,A -85,B 0,C 180,E1 -10020.38,E2 -10020.38} C_VEL
LIN {X 0,Y 417.057,Z 585.072,A -85,B 0,C 180,E1 -10022.634,E2 -10022.634} C_VEL
LIN {X 0,Y 417.344,Z 581.116,A -85,B 0,C 180,E1 -10024.93,E2 -10024.93} C_VEL
LIN {X 0,Y 417.767,Z 575.554,A -85,B 0,C 180,E1 -10027.275,E2 -10027.275} C_VEL
LIN {X 0,Y 418.354,Z 569.055,A -85,B 0,C 180,E1 -10029.397,E2 -10029.397} C_VEL
LIN {X 0,Y 419.14,Z 561.142,A -85,B 0,C 180,E1 -10031.494,E2 -10031.494} C_VEL
LIN {X 0,Y 420.076,Z 552.938,A -85,B 0,C 180,E1 -10033.311,E2 -10033.311} C_VEL
LIN {X 0,Y 421.376,Z 543.186,A -85,B 0,C 180,E1 -10035.142,E2 -10035.142} C_VEL
LIN {X 0,Y 422.806,Z 531.411,A -85,B 0,C 180,E1 -10037.003,E2 -10037.003} C_VEL
LIN {X 0,Y 424.399,Z 519.02,A -85,B 0,C 180,E1 -10038.639,E2 -10038.639} C_VEL
LIN {X 0,Y 425.92,Z 506.683,A -85,B 0,C 180,E1 -10040.022,E2 -10040.022} C_VEL
LIN {X 0,Y 427.556,Z 492.715,A -85,B 0,C 180,E1 -10041.344,E2 -10041.344} C_VEL
LIN {X 0,Y 429.116,Z 478.06,A -85,B 0,C 180,E1 -10042.499,E2 -10042.499} C_VEL
LIN {X 0,Y 430.577,Z 462.49,A -85,B 0,C 180,E1 -10043.495,E2 -10043.495} C_VEL
LIN {X 0,Y 431.776,Z 447.17,A -85,B 0,C 180,E1 -10044.268,E2 -10044.268} C_VEL
LIN {X 0,Y 432.765,Z 430.992,A -85,B 0,C 180,E1 -10044.893,E2 -10044.893} C_VEL
LIN {X 0,Y 433.512,Z 414.565,A -85,B 0,C 180,E1 -10045.339,E2 -10045.339} C_VEL
LIN {X 0,Y 437.384,Z 244.898,A -85,B 0,C 180,E1 -10048.345,E2 -10048.345} C_VEL
LIN {X 0,Y 429.532,Z 228.781,A -85,B 0,C 180,E1 -10049.35,E2 -10049.35} C_VEL
LIN {X 0,Y 421.367,Z 213.655,A -85,B 0,C 180,E1 -10050.422,E2 -10050.422} C_VEL
LIN {X 0,Y 420.022,Z 211.075,A -85,B 0,C 180,E1 -10050.628,E2 -10050.628} C_VEL
LIN {X 0,Y 418.281,Z 205.691,A -85,B 0,C 180,E1 -10051.662,E2 -10051.662} C_VEL
LIN {X 0,Y 418.271,Z 205.694,A -85,B 0,C 180,E1 -10054.095,E2 -10054.095} C_VEL
LIN {X 0,Y 418.235,Z 205.702,A -85,B 0,C 180,E1 -10057.263,E2 -10057.263} C_VEL
LIN {X 0,Y 418.286,Z 205.696,A -85,B 0,C 180,E1 -10060.364,E2 -10060.364} C_VEL
LIN {X 0,Y 418.319,Z 205.684,A -85,B 0,C 180,E1 -10063.404,E2 -10063.404} C_VEL
LIN {X 0,Y 418.348,Z 205.684,A -85,B 0,C 180,E1 -10066.999,E2 -10066.999} C_VEL
LIN {X 0,Y 418.34,Z 205.688,A -85,B 0,C 180,E1 -10070.328,E2 -10070.328} C_VEL
LIN {X 0,Y 418.493,Z 205.669,A -85,B 0,C 180,E1 -10073.248,E2 -10073.248} C_VEL
LIN {X 0,Y 418.336,Z 205.687,A -85,B 0,C 180,E1 -10075.181,E2 -10075.181} C_VEL
LIN {X 0,Y 418.541,Z 205.662,A -85,B 0,C 180,E1 -10078.075,E2 -10078.075} C_VEL
LIN {X 0,Y 418.669,Z 205.648,A -85,B 0,C 180,E1 -10080,E2 -10080} C_VEL
LIN {X 0,Y 418.499,Z 205.666,A -85,B 0,C 180,E1 -10082.887,E2 -10082.887} C_VEL
LIN {X 0,Y 418.503,Z 205.67,A -85,B 0,C 180,E1 -10085.782,E2 -10085.782} C_VEL
LIN {X 0,Y 418.378,Z 205.681,A -85,B 0,C 180,E1 -10088.695,E2 -10088.695} C_VEL
LIN {X 0,Y 418.314,Z 205.693,A -85,B 0,C 180,E1 -10091.631,E2 -10091.631} C_VEL
LIN {X 0,Y 418.301,Z 205.69,A -85,B 0,C 180,E1 -10094.597,E2 -10094.597} C_VEL
LIN {X 0,Y 418.279,Z 205.696,A -85,B 0,C 180,E1 -10097.604,E2 -10097.604} C_VEL
LIN {X 0,Y 418.249,Z 205.698,A -85,B 0,C 180,E1 -10100.663,E2 -10100.663} C_VEL
LIN {X 0,Y 418.285,Z 205.691,A -85,B 0,C 180,E1 -10103.781,E2 -10103.781} C_VEL
LIN {X 0,Y 418.311,Z 205.689,A -85,B 0,C 180,E1 -10107.07,E2 -10107.07} C_VEL
LIN {X 0,Y 418.244,Z 205.697,A -85,B 0,C 180,E1 -10110.272,E2 -10110.272} C_VEL
LIN {X 0,Y 418.233,Z 205.698,A -85,B 0,C 180,E1 -10113.678,E2 -10113.678} C_VEL
LIN {X 0,Y 418.24,Z 205.702,A -85,B 0,C 180,E1 -10117.224,E2 -10117.224} C_VEL
LIN {X 0,Y 418.244,Z 205.699,A -85,B 0,C 180,E1 -10119.682,E2 -10119.682} C_VEL
